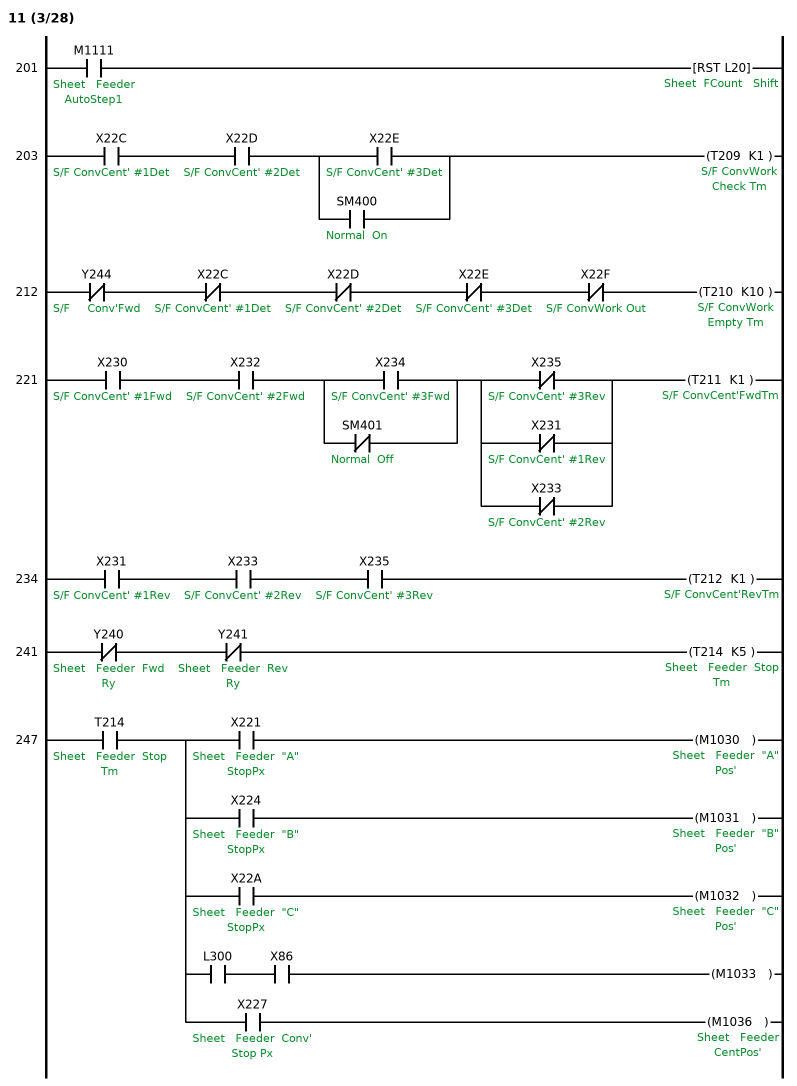
201   LD      M1111  ; Sheet   Feeder  AutoStep1
      RST     L20  ; Sheet  FCount   Shift
203   LD      X22C  ; S/F ConvCent' #1Det
      AND     X22D  ; S/F ConvCent' #2Det
      LD      X22E  ; S/F ConvCent' #3Det
      OR      SM400  ; Normal  On
      ANB
      OUT     T209 K1  ; S/F ConvWork    Check Tm
212   LDI     Y244  ; S/F     Conv'Fwd
      ANI     X22C  ; S/F ConvCent' #1Det
      ANI     X22D  ; S/F ConvCent' #2Det
      ANI     X22E  ; S/F ConvCent' #3Det
      ANI     X22F  ; S/F ConvWork Out
      OUT     T210 K10  ; S/F ConvWork    Empty Tm
221   LD      X230  ; S/F ConvCent' #1Fwd
      AND     X232  ; S/F ConvCent' #2Fwd
      LD      X234  ; S/F ConvCent' #3Fwd
      ORI     SM401  ; Normal  Off
      ANB
      LDI     X235  ; S/F ConvCent' #3Rev
      ORI     X231  ; S/F ConvCent' #1Rev
      ORI     X233  ; S/F ConvCent' #2Rev
      ANB
      OUT     T211 K1  ; S/F ConvCent'FwdTm
234   LD      X231  ; S/F ConvCent' #1Rev
      AND     X233  ; S/F ConvCent' #2Rev
      AND     X235  ; S/F ConvCent' #3Rev
      OUT     T212 K1  ; S/F ConvCent'RevTm
241   LDI     Y240  ; Sheet   Feeder  Fwd Ry
      ANI     Y241  ; Sheet   Feeder  Rev Ry
      OUT     T214 K5  ; Sheet   Feeder  Stop Tm
247   LD      T214  ; Sheet   Feeder  Stop Tm
      MPS
      AND     X221  ; Sheet   Feeder  "A" StopPx
      OUT     M1030  ; Sheet   Feeder  "A" Pos'
      MRD
      AND     X224  ; Sheet   Feeder  "B" StopPx
      OUT     M1031  ; Sheet   Feeder  "B" Pos'
      MRD
      AND     X22A  ; Sheet   Feeder  "C" StopPx
      OUT     M1032  ; Sheet   Feeder  "C" Pos'
      MRD
      AND     L300
      AND     X86
      OUT     M1033
      MPP
      AND     X227  ; Sheet   Feeder  Conv'   Stop Px
      OUT     M1036  ; Sheet   Feeder  CentPos'
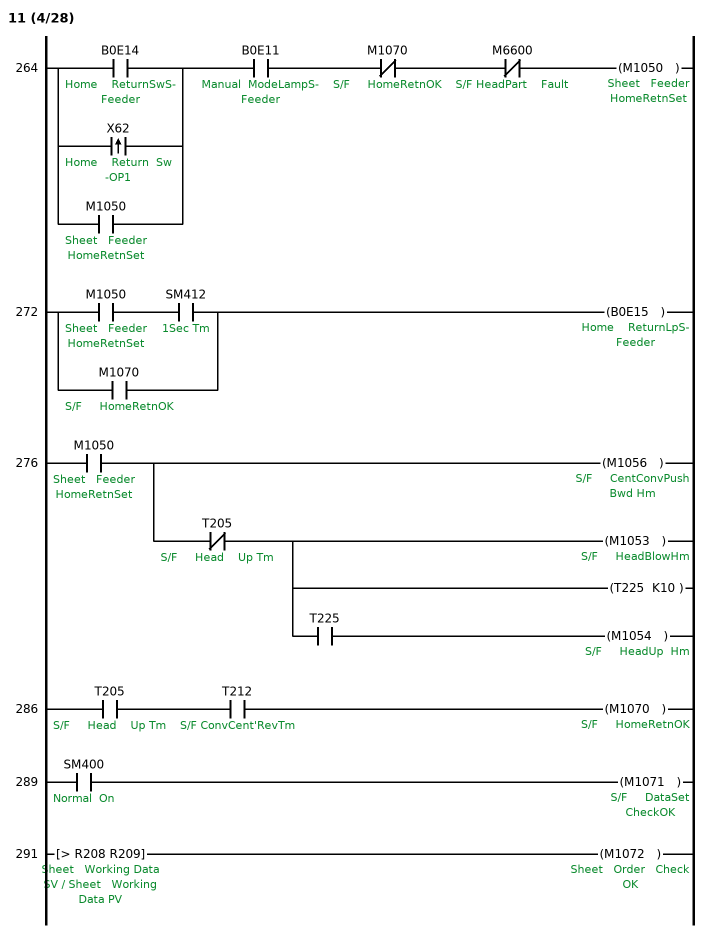
264   LD      B0E14  ; Home    ReturnSwS-Feeder
      ORP     X62  ; Home    Return  Sw -OP1
      OR      M1050  ; Sheet   Feeder  HomeRetnSet
      AND     B0E11  ; Manual  ModeLampS-Feeder
      ANI     M1070  ; S/F     HomeRetnOK
      ANI     M6600  ; S/F HeadPart    Fault
      OUT     M1050  ; Sheet   Feeder  HomeRetnSet
272   LD      M1050  ; Sheet   Feeder  HomeRetnSet
      AND     SM412  ; 1Sec Tm
      OR      M1070  ; S/F     HomeRetnOK
      OUT     B0E15  ; Home    ReturnLpS-Feeder
276   LD      M1050  ; Sheet   Feeder  HomeRetnSet
      OUT     M1056  ; S/F     CentConvPushBwd Hm
      ANI     T205  ; S/F     Head    Up Tm
      OUT     M1053  ; S/F     HeadBlowHm
      OUT     T225 K10
      AND     T225
      OUT     M1054  ; S/F     HeadUp  Hm
286   LD      T205  ; S/F     Head    Up Tm
      AND     T212  ; S/F ConvCent'RevTm
      OUT     M1070  ; S/F     HomeRetnOK
289   LD      SM400  ; Normal  On
      OUT     M1071  ; S/F     DataSet CheckOK
291   LD>     R208 R209  ; Sheet   Working Data SV / Sheet   Working Data PV
      OUT     M1072  ; Sheet   Order   Check OK
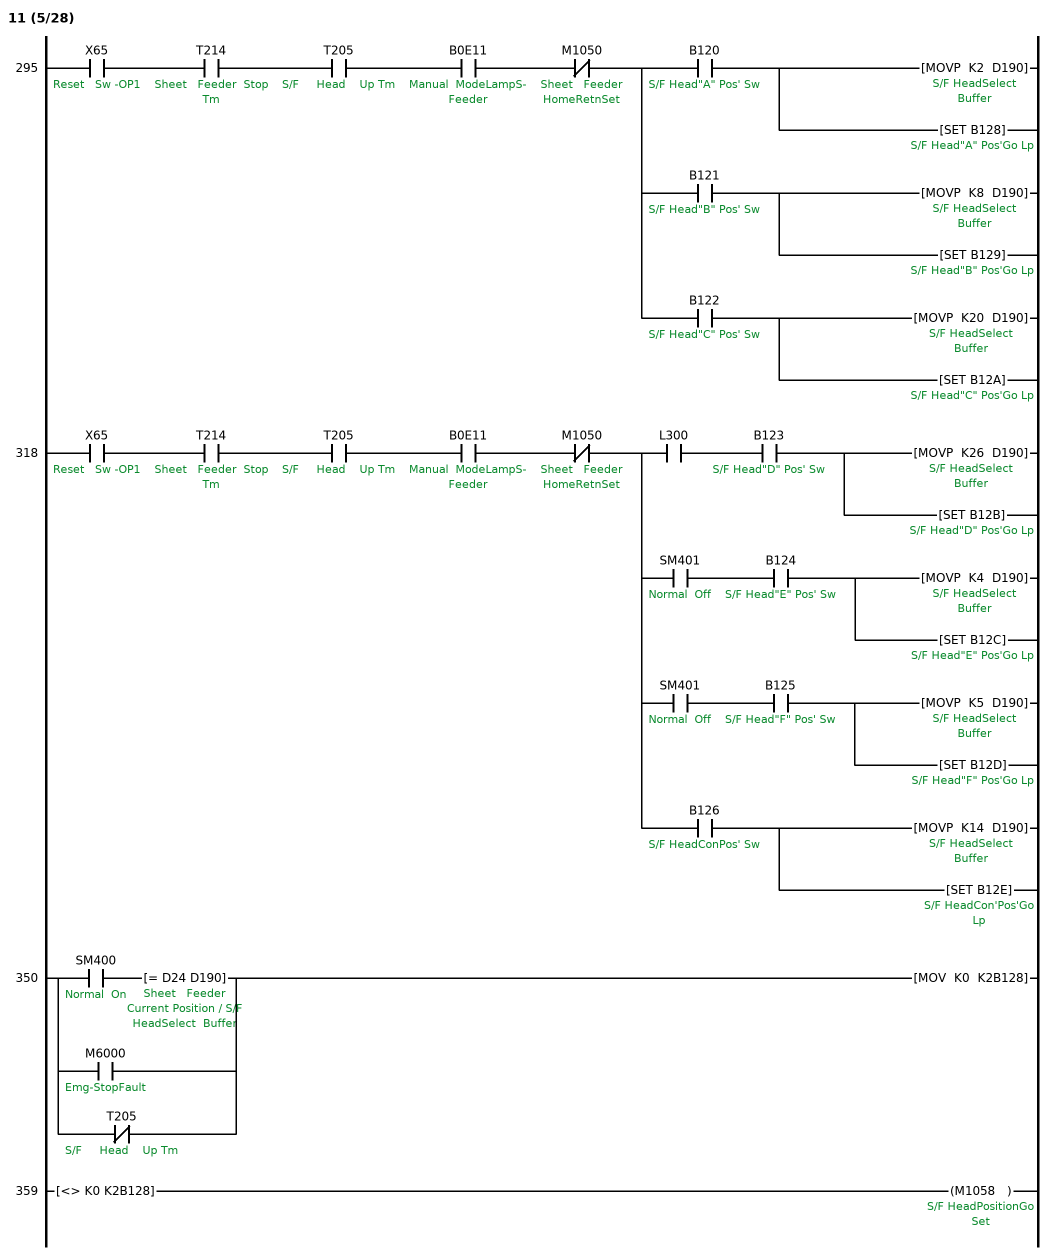
295   LD      X65  ; Reset   Sw -OP1
      AND     T214  ; Sheet   Feeder  Stop Tm
      AND     T205  ; S/F     Head    Up Tm
      AND     B0E11  ; Manual  ModeLampS-Feeder
      ANI     M1050  ; Sheet   Feeder  HomeRetnSet
      MPS
      AND     B120  ; S/F Head"A" Pos' Sw
      MOVP    K2 D190  ; S/F HeadSelect  Buffer
      SET     B128  ; S/F Head"A" Pos'Go Lp
      MRD
      AND     B121  ; S/F Head"B" Pos' Sw
      MOVP    K8 D190
      SET     B129  ; S/F Head"B" Pos'Go Lp
      MPP
      AND     B122  ; S/F Head"C" Pos' Sw
      MOVP    K20 D190
      SET     B12A  ; S/F Head"C" Pos'Go Lp
318   LD      X65  ; Reset   Sw -OP1
      AND     T214  ; Sheet   Feeder  Stop Tm
      AND     T205  ; S/F     Head    Up Tm
      AND     B0E11  ; Manual  ModeLampS-Feeder
      ANI     M1050  ; Sheet   Feeder  HomeRetnSet
      MPS
      AND     L300
      AND     B123  ; S/F Head"D" Pos' Sw
      MOVP    K26 D190
      SET     B12B  ; S/F Head"D" Pos'Go Lp
      MRD
      AND     SM401  ; Normal  Off
      AND     B124  ; S/F Head"E" Pos' Sw
      MOVP    K4 D190
      SET     B12C  ; S/F Head"E" Pos'Go Lp
      MRD
      AND     SM401  ; Normal  Off
      AND     B125  ; S/F Head"F" Pos' Sw
      MOVP    K5 D190
      SET     B12D  ; S/F Head"F" Pos'Go Lp
      MPP
      AND     B126  ; S/F HeadConPos' Sw
      MOVP    K14 D190
      SET     B12E  ; S/F HeadCon'Pos'Go Lp
350   LD      SM400  ; Normal  On
      AND=    D24 D190  ; Sheet   Feeder  Current Position / S/F HeadSelect  Buffer
      OR      M6000  ; Emg-StopFault
      ORI     T205  ; S/F     Head    Up Tm
      MOV     K0 K2B128
359   LD<>    K0 K2B128  ; S/F Head"A" Pos'Go Lp
      OUT     M1058  ; S/F HeadPositionGo Set
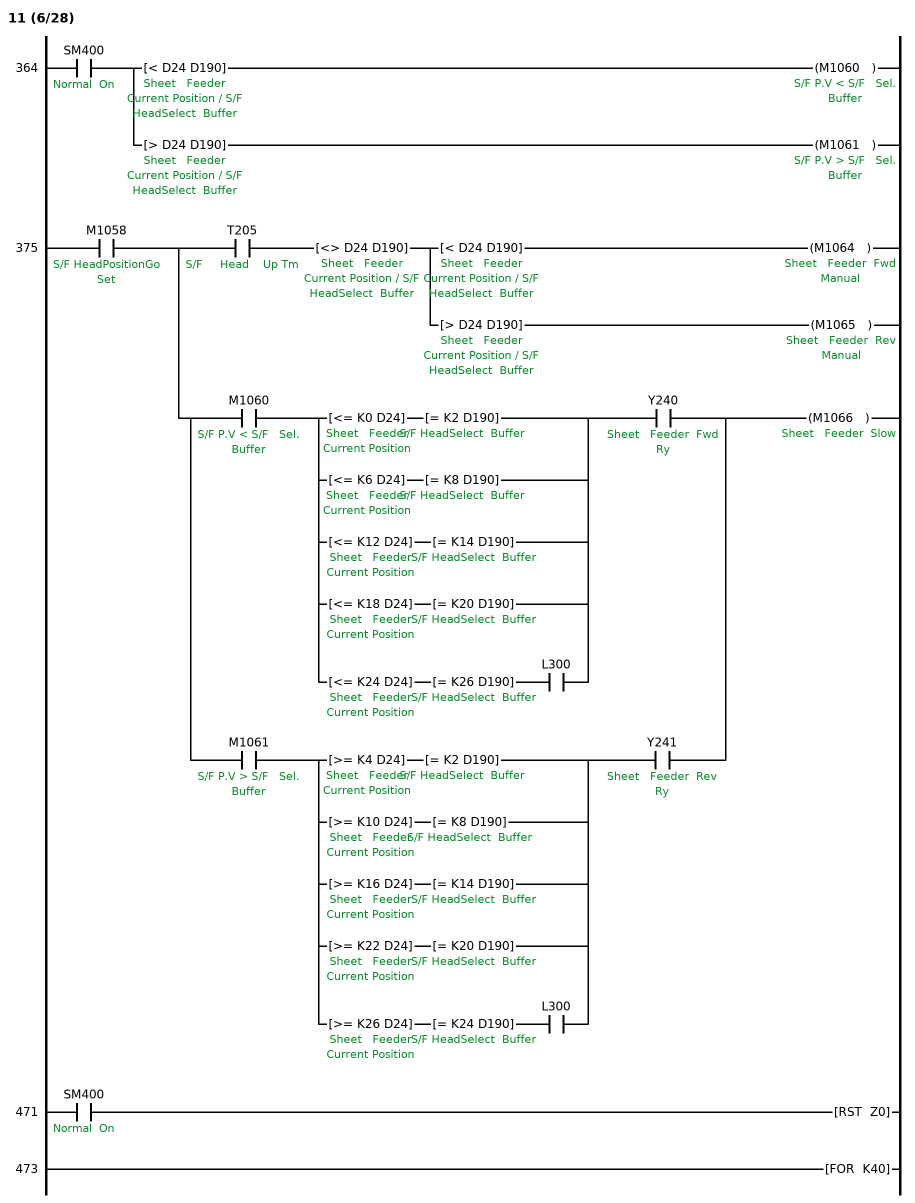
364   LD      SM400  ; Normal  On
      MPS
      AND<    D24 D190  ; Sheet   Feeder  Current Position / S/F HeadSelect  Buffer
      OUT     M1060  ; S/F P.V < S/F   Sel.    Buffer
      MPP
      AND>    D24 D190  ; Sheet   Feeder  Current Position / S/F HeadSelect  Buffer
      OUT     M1061  ; S/F P.V > S/F   Sel.    Buffer
375   LD      M1058  ; S/F HeadPositionGo Set
      MPS
      AND     T205  ; S/F     Head    Up Tm
      AND<>   D24 D190  ; Sheet   Feeder  Current Position / S/F HeadSelect  Buffer
      MPS
      AND<    D24 D190  ; Sheet   Feeder  Current Position / S/F HeadSelect  Buffer
      OUT     M1064  ; Sheet   Feeder  Fwd     Manual
      MPP
      AND>    D24 D190  ; Sheet   Feeder  Current Position / S/F HeadSelect  Buffer
      OUT     M1065  ; Sheet   Feeder  Rev     Manual
      MPP
      LD      M1060  ; S/F P.V < S/F   Sel.    Buffer
      LD<=    K0 D24  ; Sheet   Feeder  Current Position
      AND=    K2 D190  ; S/F HeadSelect  Buffer
      LD<=    K6 D24  ; Sheet   Feeder  Current Position
      AND=    K8 D190  ; S/F HeadSelect  Buffer
      ORB
      LD<=    K12 D24  ; Sheet   Feeder  Current Position
      AND=    K14 D190  ; S/F HeadSelect  Buffer
      ORB
      LD<=    K18 D24  ; Sheet   Feeder  Current Position
      AND=    K20 D190  ; S/F HeadSelect  Buffer
      ORB
      LD<=    K24 D24  ; Sheet   Feeder  Current Position
      AND=    K26 D190  ; S/F HeadSelect  Buffer
      AND     L300
      ORB
      ANB
      AND     Y240  ; Sheet   Feeder  Fwd Ry
      LD      M1061  ; S/F P.V > S/F   Sel.    Buffer
      LD>=    K4 D24  ; Sheet   Feeder  Current Position
      AND=    K2 D190  ; S/F HeadSelect  Buffer
      LD>=    K10 D24  ; Sheet   Feeder  Current Position
      AND=    K8 D190  ; S/F HeadSelect  Buffer
      ORB
      LD>=    K16 D24  ; Sheet   Feeder  Current Position
      AND=    K14 D190  ; S/F HeadSelect  Buffer
      ORB
      LD>=    K22 D24  ; Sheet   Feeder  Current Position
      AND=    K20 D190  ; S/F HeadSelect  Buffer
      ORB
      LD>=    K26 D24  ; Sheet   Feeder  Current Position
      AND=    K24 D190  ; S/F HeadSelect  Buffer
      AND     L300
      ORB
      ANB
      AND     Y241  ; Sheet   Feeder  Rev Ry
      ORB
      ANB
      OUT     M1066  ; Sheet   Feeder  Slow
471   LD      SM400  ; Normal  On
      RST     Z0
473   FOR     K40
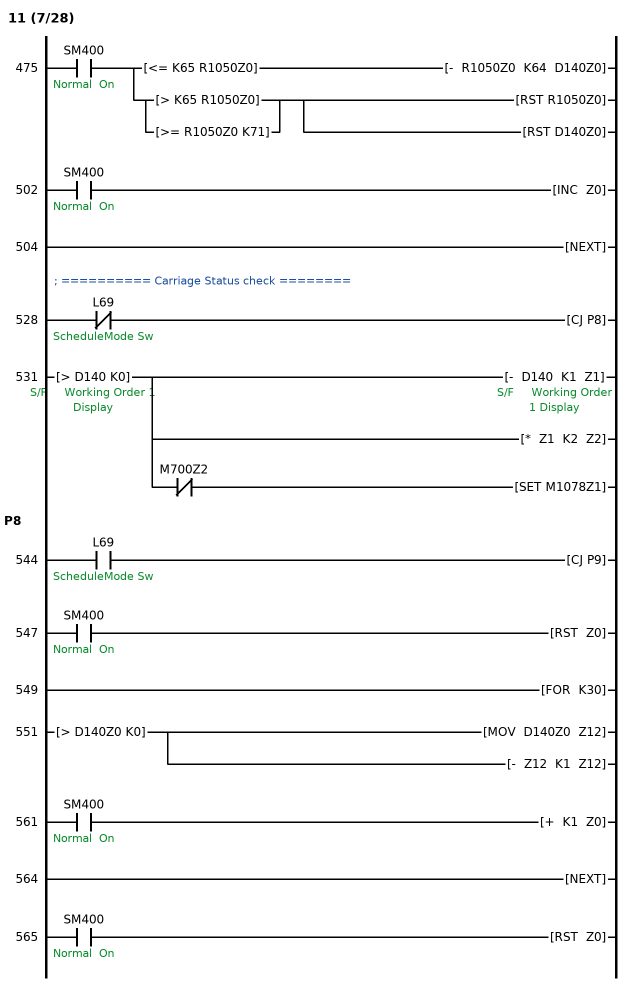
475   LD      SM400  ; Normal  On
      MPS
      AND<=   K65 R1050Z0
      -       R1050Z0 K64 D140Z0
      MPP
      LD>     K65 R1050Z0
      OR>=    R1050Z0 K71
      ANB
      RST     R1050Z0
      RST     D140Z0
502   LD      SM400  ; Normal  On
      INC     Z0
504   NEXT
; ========== Carriage Status check ========
528   LDI     L69  ; ScheduleMode Sw
      CJ      P8
531   LD>     D140 K0  ; S/F     Working Order 1 Display
      -       D140 K1 Z1
      *       Z1 K2 Z2
      ANI     M700Z2
      SET     M1078Z1
      P8
544   LD      L69  ; ScheduleMode Sw
      CJ      P9
547   LD      SM400  ; Normal  On
      RST     Z0
549   FOR     K30
551   LD>     D140Z0 K0
      MOV     D140Z0 Z12
      -       Z12 K1 Z12
561   LD      SM400  ; Normal  On
      +       K1 Z0
564   NEXT
565   LD      SM400  ; Normal  On
      RST     Z0
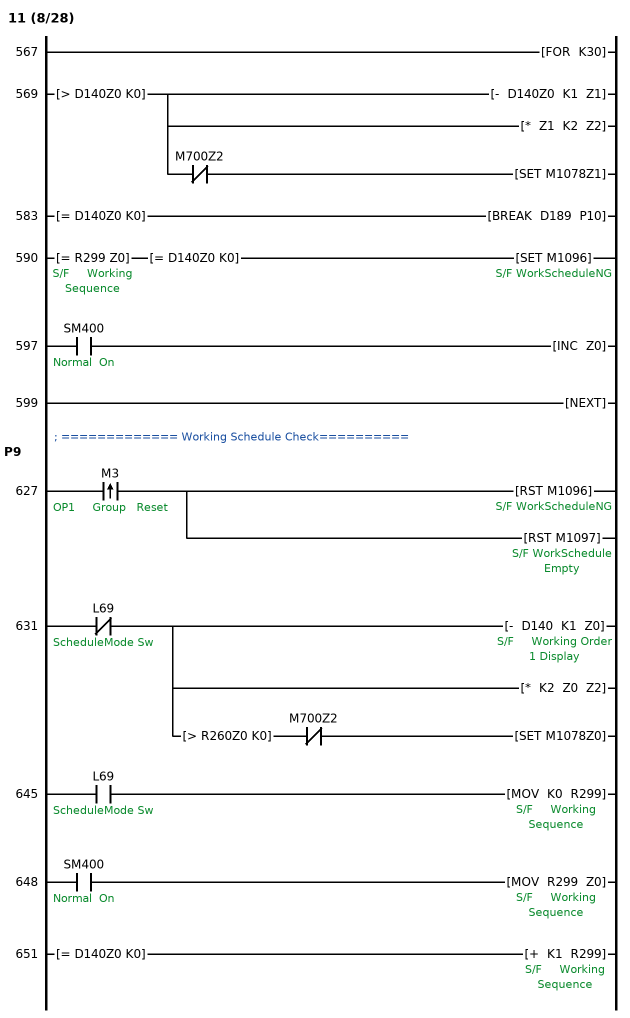
567   FOR     K30
569   LD>     D140Z0 K0
      -       D140Z0 K1 Z1
      *       Z1 K2 Z2
      ANI     M700Z2
      SET     M1078Z1
583   LD=     D140Z0 K0
      BREAK   D189 P10
590   LD=     R299 Z0  ; S/F     Working Sequence
      AND=    D140Z0 K0
      SET     M1096  ; S/F WorkScheduleNG
597   LD      SM400  ; Normal  On
      INC     Z0
599   NEXT
      P10
; ============= Working Schedule Check==========
      P9
627   LDP     M3  ; OP1     Group   Reset
      RST     M1096  ; S/F WorkScheduleNG
      RST     M1097  ; S/F WorkScheduleEmpty
631   LDI     L69  ; ScheduleMode Sw
      -       D140 K1 Z0
      *       K2 Z0 Z2
      AND>    R260Z0 K0
      ANI     M700Z2
      SET     M1078Z0
645   LD      L69  ; ScheduleMode Sw
      MOV     K0 R299
648   LD      SM400  ; Normal  On
      MOV     R299 Z0
651   LD=     D140Z0 K0
      +       K1 R299
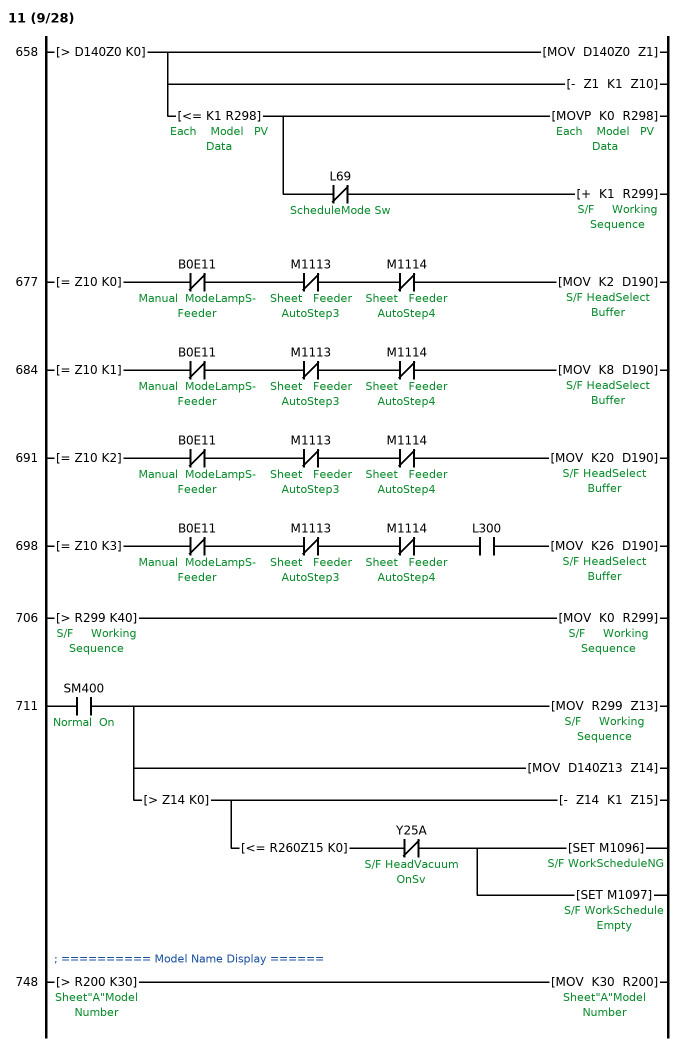
658   LD>     D140Z0 K0
      MOV     D140Z0 Z1
      -       Z1 K1 Z10
      AND<=   K1 R298  ; Each    Model   PV Data
      MOVP    K0 R298
      ANI     L69  ; ScheduleMode Sw
      +       K1 R299
677   LD=     Z10 K0
      ANI     B0E11  ; Manual  ModeLampS-Feeder
      ANI     M1113  ; Sheet   Feeder  AutoStep3
      ANI     M1114  ; Sheet   Feeder  AutoStep4
      MOV     K2 D190
684   LD=     Z10 K1
      ANI     B0E11  ; Manual  ModeLampS-Feeder
      ANI     M1113  ; Sheet   Feeder  AutoStep3
      ANI     M1114  ; Sheet   Feeder  AutoStep4
      MOV     K8 D190
691   LD=     Z10 K2
      ANI     B0E11  ; Manual  ModeLampS-Feeder
      ANI     M1113  ; Sheet   Feeder  AutoStep3
      ANI     M1114  ; Sheet   Feeder  AutoStep4
      MOV     K20 D190
698   LD=     Z10 K3
      ANI     B0E11  ; Manual  ModeLampS-Feeder
      ANI     M1113  ; Sheet   Feeder  AutoStep3
      ANI     M1114  ; Sheet   Feeder  AutoStep4
      AND     L300
      MOV     K26 D190
706   LD>     R299 K40  ; S/F     Working Sequence
      MOV     K0 R299
711   LD      SM400  ; Normal  On
      MOV     R299 Z13
      MOV     D140Z13 Z14
      AND>    Z14 K0
      -       Z14 K1 Z15
      AND<=   R260Z15 K0
      ANI     Y25A  ; S/F HeadVacuum  OnSv
      SET     M1096  ; S/F WorkScheduleNG
      SET     M1097  ; S/F WorkScheduleEmpty
; ========== Model Name Display ======
748   LD>     R200 K30  ; Sheet"A"Model   Number
      MOV     K30 R200
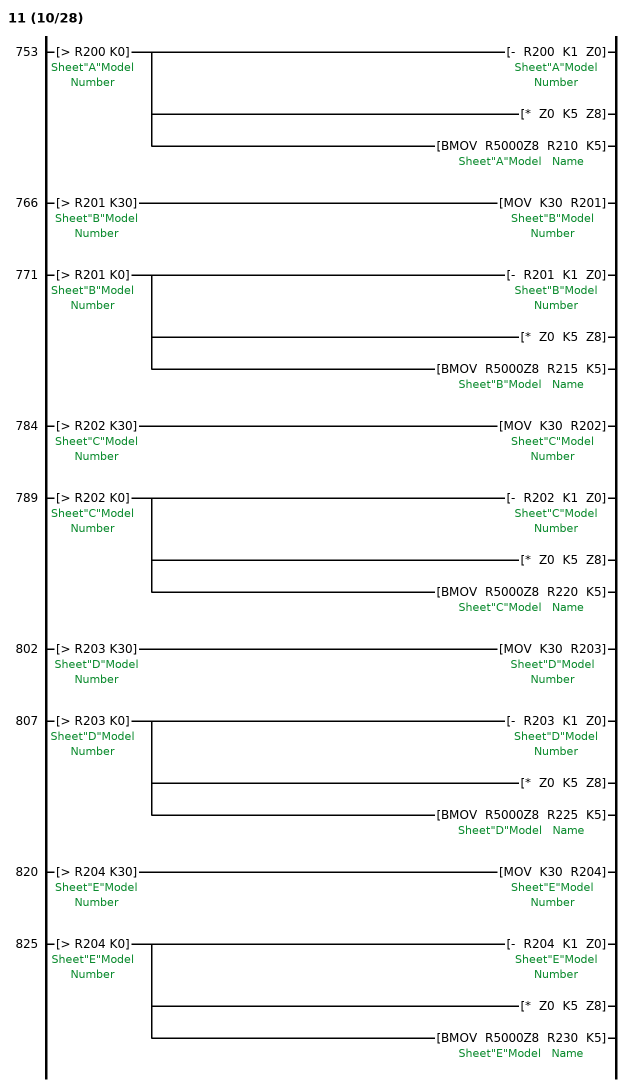
753   LD>     R200 K0  ; Sheet"A"Model   Number
      -       R200 K1 Z0
      *       Z0 K5 Z8
      BMOV    R5000Z8 R210 K5  ; Sheet"A"Model   Name
766   LD>     R201 K30  ; Sheet"B"Model   Number
      MOV     K30 R201
771   LD>     R201 K0  ; Sheet"B"Model   Number
      -       R201 K1 Z0
      *       Z0 K5 Z8
      BMOV    R5000Z8 R215 K5  ; Sheet"B"Model   Name
784   LD>     R202 K30  ; Sheet"C"Model   Number
      MOV     K30 R202
789   LD>     R202 K0  ; Sheet"C"Model   Number
      -       R202 K1 Z0
      *       Z0 K5 Z8
      BMOV    R5000Z8 R220 K5  ; Sheet"C"Model   Name
802   LD>     R203 K30  ; Sheet"D"Model   Number
      MOV     K30 R203
807   LD>     R203 K0  ; Sheet"D"Model   Number
      -       R203 K1 Z0
      *       Z0 K5 Z8
      BMOV    R5000Z8 R225 K5  ; Sheet"D"Model   Name
820   LD>     R204 K30  ; Sheet"E"Model   Number
      MOV     K30 R204
825   LD>     R204 K0  ; Sheet"E"Model   Number
      -       R204 K1 Z0
      *       Z0 K5 Z8
      BMOV    R5000Z8 R230 K5  ; Sheet"E"Model   Name
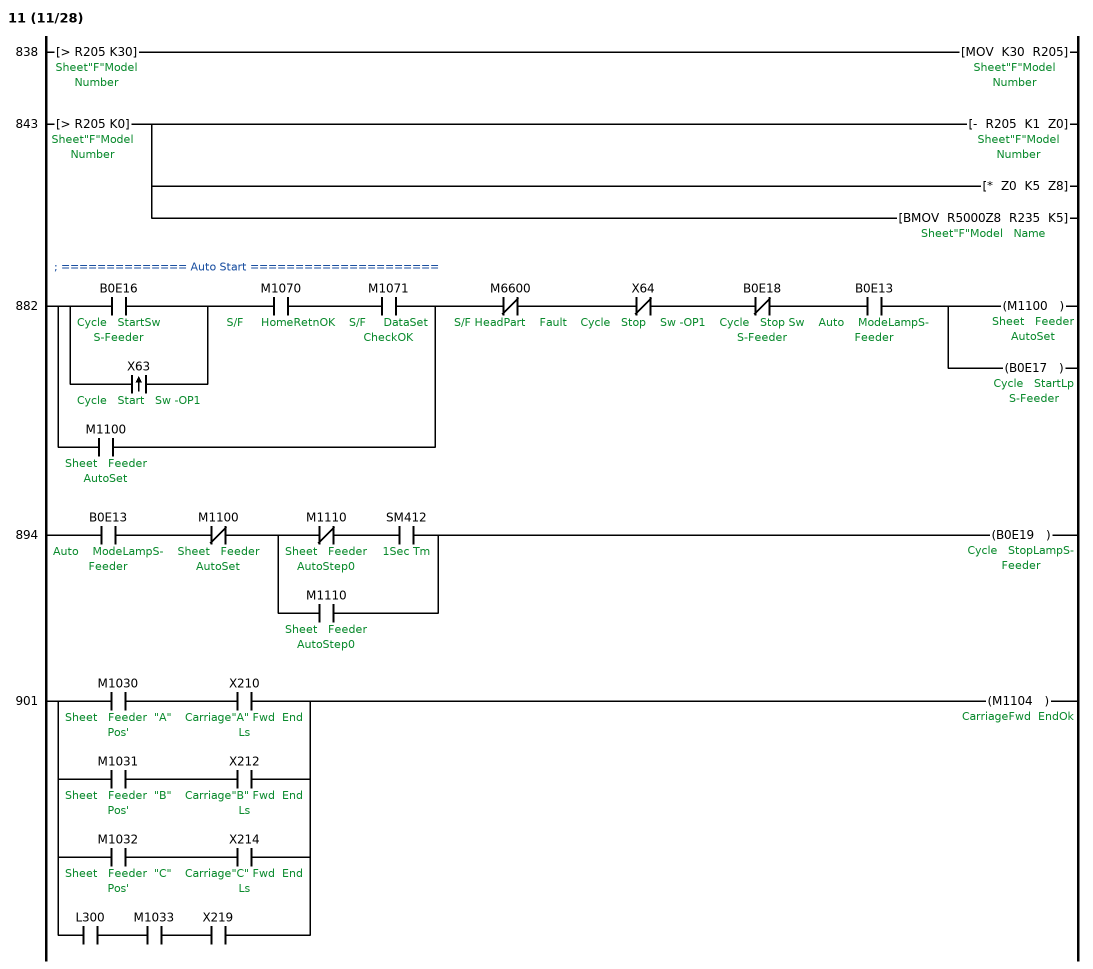
838   LD>     R205 K30  ; Sheet"F"Model   Number
      MOV     K30 R205
843   LD>     R205 K0  ; Sheet"F"Model   Number
      -       R205 K1 Z0
      *       Z0 K5 Z8
      BMOV    R5000Z8 R235 K5  ; Sheet"F"Model   Name
; ============== Auto Start =====================
882   LD      B0E16  ; Cycle   StartSw S-Feeder
      ORP     X63  ; Cycle   Start   Sw -OP1
      AND     M1070  ; S/F     HomeRetnOK
      AND     M1071  ; S/F     DataSet CheckOK
      OR      M1100  ; Sheet   Feeder  AutoSet
      ANI     M6600  ; S/F HeadPart    Fault
      ANI     X64  ; Cycle   Stop    Sw -OP1
      ANI     B0E18  ; Cycle   Stop Sw S-Feeder
      AND     B0E13  ; Auto    ModeLampS-Feeder
      OUT     M1100  ; Sheet   Feeder  AutoSet
      OUT     B0E17  ; Cycle   StartLp S-Feeder
894   LD      B0E13  ; Auto    ModeLampS-Feeder
      ANI     M1100  ; Sheet   Feeder  AutoSet
      LDI     M1110  ; Sheet   Feeder  AutoStep0
      AND     SM412  ; 1Sec Tm
      OR      M1110  ; Sheet   Feeder  AutoStep0
      ANB
      OUT     B0E19  ; Cycle   StopLampS-Feeder
901   LD      M1030  ; Sheet   Feeder  "A" Pos'
      AND     X210  ; Carriage"A" Fwd  End Ls
      LD      M1031  ; Sheet   Feeder  "B" Pos'
      AND     X212  ; Carriage"B" Fwd  End Ls
      ORB
      LD      M1032  ; Sheet   Feeder  "C" Pos'
      AND     X214  ; Carriage"C" Fwd  End Ls
      ORB
      LD      L300
      AND     M1033
      AND     X219
      ORB
      OUT     M1104  ; CarriageFwd  EndOk
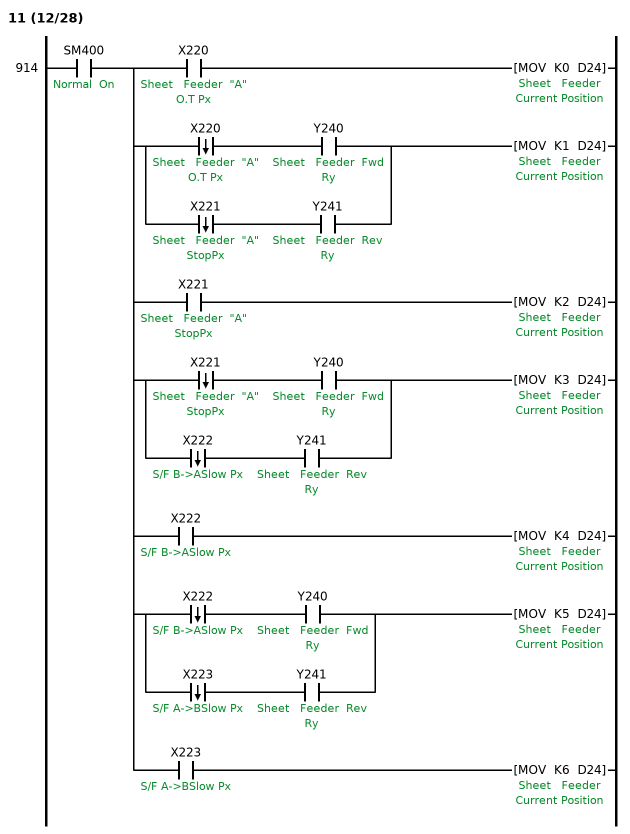
914   LD      SM400  ; Normal  On
      MPS
      AND     X220  ; Sheet   Feeder  "A" O.T Px
      MOV     K0 D24
      MRD
      LDF     X220  ; Sheet   Feeder  "A" O.T Px
      AND     Y240  ; Sheet   Feeder  Fwd Ry
      LDF     X221  ; Sheet   Feeder  "A" StopPx
      AND     Y241  ; Sheet   Feeder  Rev Ry
      ORB
      ANB
      MOV     K1 D24
      MRD
      AND     X221  ; Sheet   Feeder  "A" StopPx
      MOV     K2 D24
      MRD
      LDF     X221  ; Sheet   Feeder  "A" StopPx
      AND     Y240  ; Sheet   Feeder  Fwd Ry
      LDF     X222  ; S/F B->ASlow Px
      AND     Y241  ; Sheet   Feeder  Rev Ry
      ORB
      ANB
      MOV     K3 D24
      MRD
      AND     X222  ; S/F B->ASlow Px
      MOV     K4 D24
      MRD
      LDF     X222  ; S/F B->ASlow Px
      AND     Y240  ; Sheet   Feeder  Fwd Ry
      LDF     X223  ; S/F A->BSlow Px
      AND     Y241  ; Sheet   Feeder  Rev Ry
      ORB
      ANB
      MOV     K5 D24
      MPP
      AND     X223  ; S/F A->BSlow Px
      MOV     K6 D24
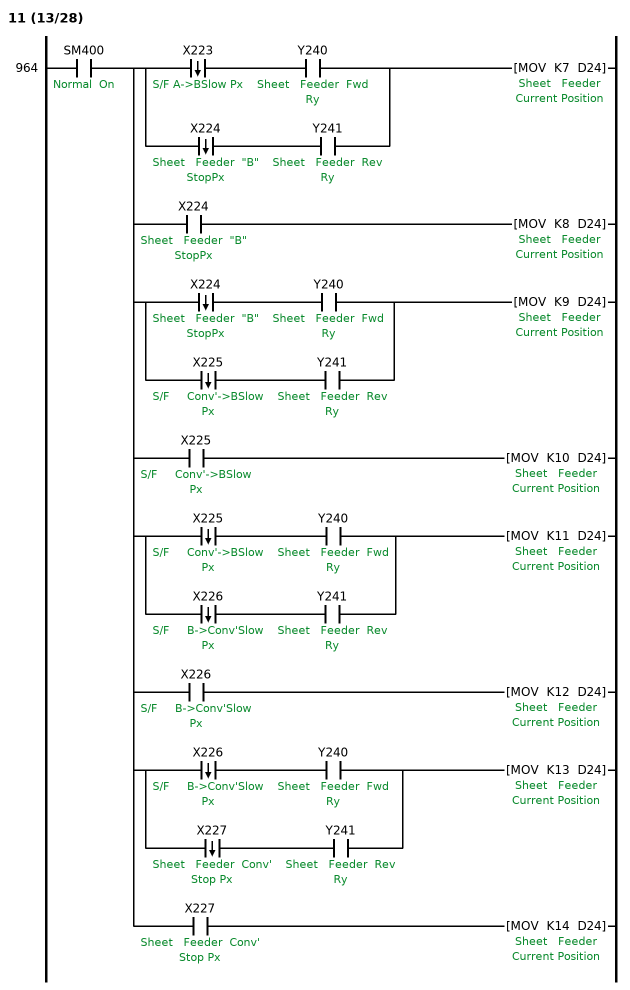
964   LD      SM400  ; Normal  On
      MPS
      LDF     X223  ; S/F A->BSlow Px
      AND     Y240  ; Sheet   Feeder  Fwd Ry
      LDF     X224  ; Sheet   Feeder  "B" StopPx
      AND     Y241  ; Sheet   Feeder  Rev Ry
      ORB
      ANB
      MOV     K7 D24
      MRD
      AND     X224  ; Sheet   Feeder  "B" StopPx
      MOV     K8 D24
      MRD
      LDF     X224  ; Sheet   Feeder  "B" StopPx
      AND     Y240  ; Sheet   Feeder  Fwd Ry
      LDF     X225  ; S/F     Conv'->BSlow Px
      AND     Y241  ; Sheet   Feeder  Rev Ry
      ORB
      ANB
      MOV     K9 D24
      MRD
      AND     X225  ; S/F     Conv'->BSlow Px
      MOV     K10 D24
      MRD
      LDF     X225  ; S/F     Conv'->BSlow Px
      AND     Y240  ; Sheet   Feeder  Fwd Ry
      LDF     X226  ; S/F     B->Conv'Slow Px
      AND     Y241  ; Sheet   Feeder  Rev Ry
      ORB
      ANB
      MOV     K11 D24
      MRD
      AND     X226  ; S/F     B->Conv'Slow Px
      MOV     K12 D24
      MRD
      LDF     X226  ; S/F     B->Conv'Slow Px
      AND     Y240  ; Sheet   Feeder  Fwd Ry
      LDF     X227  ; Sheet   Feeder  Conv'   Stop Px
      AND     Y241  ; Sheet   Feeder  Rev Ry
      ORB
      ANB
      MOV     K13 D24
      MPP
      AND     X227  ; Sheet   Feeder  Conv'   Stop Px
      MOV     K14 D24
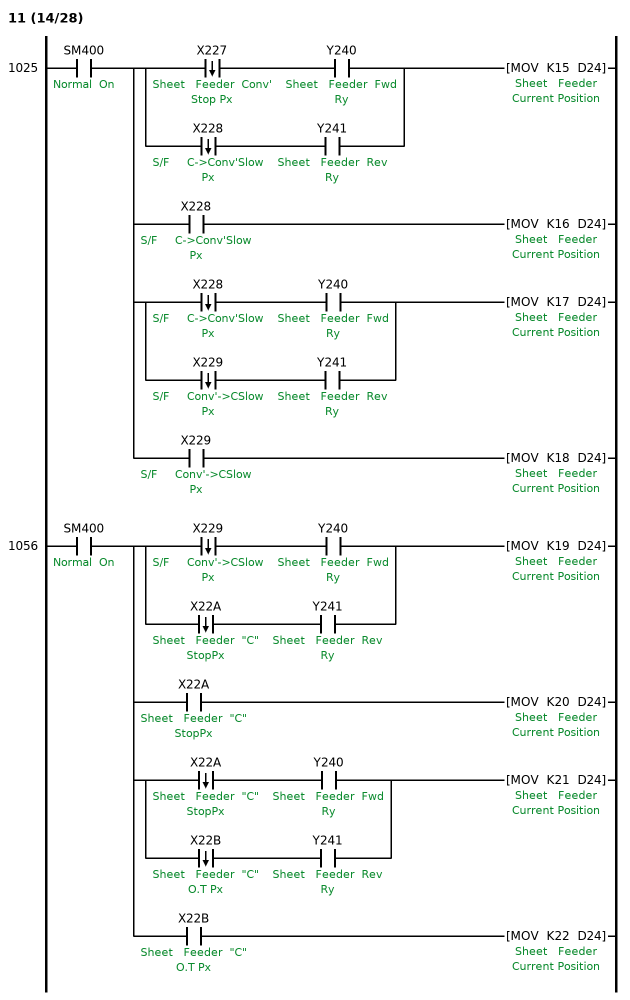
1025  LD      SM400  ; Normal  On
      MPS
      LDF     X227  ; Sheet   Feeder  Conv'   Stop Px
      AND     Y240  ; Sheet   Feeder  Fwd Ry
      LDF     X228  ; S/F     C->Conv'Slow Px
      AND     Y241  ; Sheet   Feeder  Rev Ry
      ORB
      ANB
      MOV     K15 D24
      MRD
      AND     X228  ; S/F     C->Conv'Slow Px
      MOV     K16 D24
      MRD
      LDF     X228  ; S/F     C->Conv'Slow Px
      AND     Y240  ; Sheet   Feeder  Fwd Ry
      LDF     X229  ; S/F     Conv'->CSlow Px
      AND     Y241  ; Sheet   Feeder  Rev Ry
      ORB
      ANB
      MOV     K17 D24
      MPP
      AND     X229  ; S/F     Conv'->CSlow Px
      MOV     K18 D24
1056  LD      SM400  ; Normal  On
      MPS
      LDF     X229  ; S/F     Conv'->CSlow Px
      AND     Y240  ; Sheet   Feeder  Fwd Ry
      LDF     X22A  ; Sheet   Feeder  "C" StopPx
      AND     Y241  ; Sheet   Feeder  Rev Ry
      ORB
      ANB
      MOV     K19 D24
      MRD
      AND     X22A  ; Sheet   Feeder  "C" StopPx
      MOV     K20 D24
      MRD
      LDF     X22A  ; Sheet   Feeder  "C" StopPx
      AND     Y240  ; Sheet   Feeder  Fwd Ry
      LDF     X22B  ; Sheet   Feeder  "C" O.T Px
      AND     Y241  ; Sheet   Feeder  Rev Ry
      ORB
      ANB
      MOV     K21 D24
      MPP
      AND     X22B  ; Sheet   Feeder  "C" O.T Px
      MOV     K22 D24
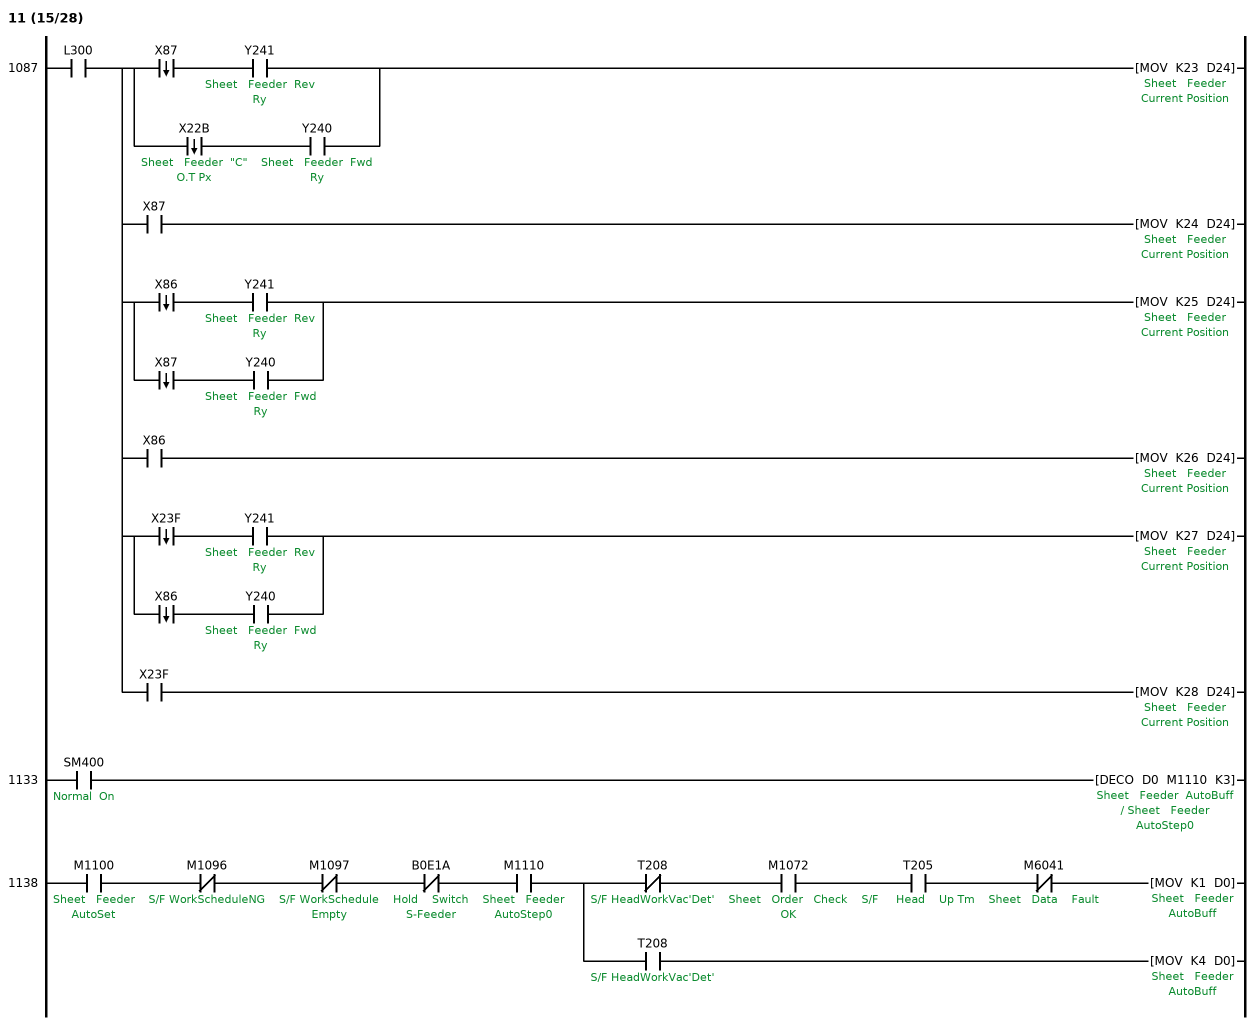
1087  LD      L300
      MPS
      LDF     X87
      AND     Y241  ; Sheet   Feeder  Rev Ry
      LDF     X22B  ; Sheet   Feeder  "C" O.T Px
      AND     Y240  ; Sheet   Feeder  Fwd Ry
      ORB
      ANB
      MOV     K23 D24
      MRD
      AND     X87
      MOV     K24 D24
      MRD
      LDF     X86
      AND     Y241  ; Sheet   Feeder  Rev Ry
      LDF     X87
      AND     Y240  ; Sheet   Feeder  Fwd Ry
      ORB
      ANB
      MOV     K25 D24
      MRD
      AND     X86
      MOV     K26 D24
      MRD
      LDF     X23F
      AND     Y241  ; Sheet   Feeder  Rev Ry
      LDF     X86
      AND     Y240  ; Sheet   Feeder  Fwd Ry
      ORB
      ANB
      MOV     K27 D24
      MPP
      AND     X23F
      MOV     K28 D24
1133  LD      SM400  ; Normal  On
      DECO    D0 M1110 K3  ; Sheet   Feeder  AutoBuff
1138  LD      M1100  ; Sheet   Feeder  AutoSet
      ANI     M1096  ; S/F WorkScheduleNG
      ANI     M1097  ; S/F WorkScheduleEmpty
      ANI     B0E1A  ; Hold    Switch  S-Feeder
      AND     M1110  ; Sheet   Feeder  AutoStep0
      MPS
      ANI     T208  ; S/F HeadWorkVac'Det'
      AND     M1072  ; Sheet   Order   Check OK
      AND     T205  ; S/F     Head    Up Tm
      ANI     M6041  ; Sheet   Data    Fault
      MOV     K1 D0
      MPP
      AND     T208  ; S/F HeadWorkVac'Det'
      MOV     K4 D0
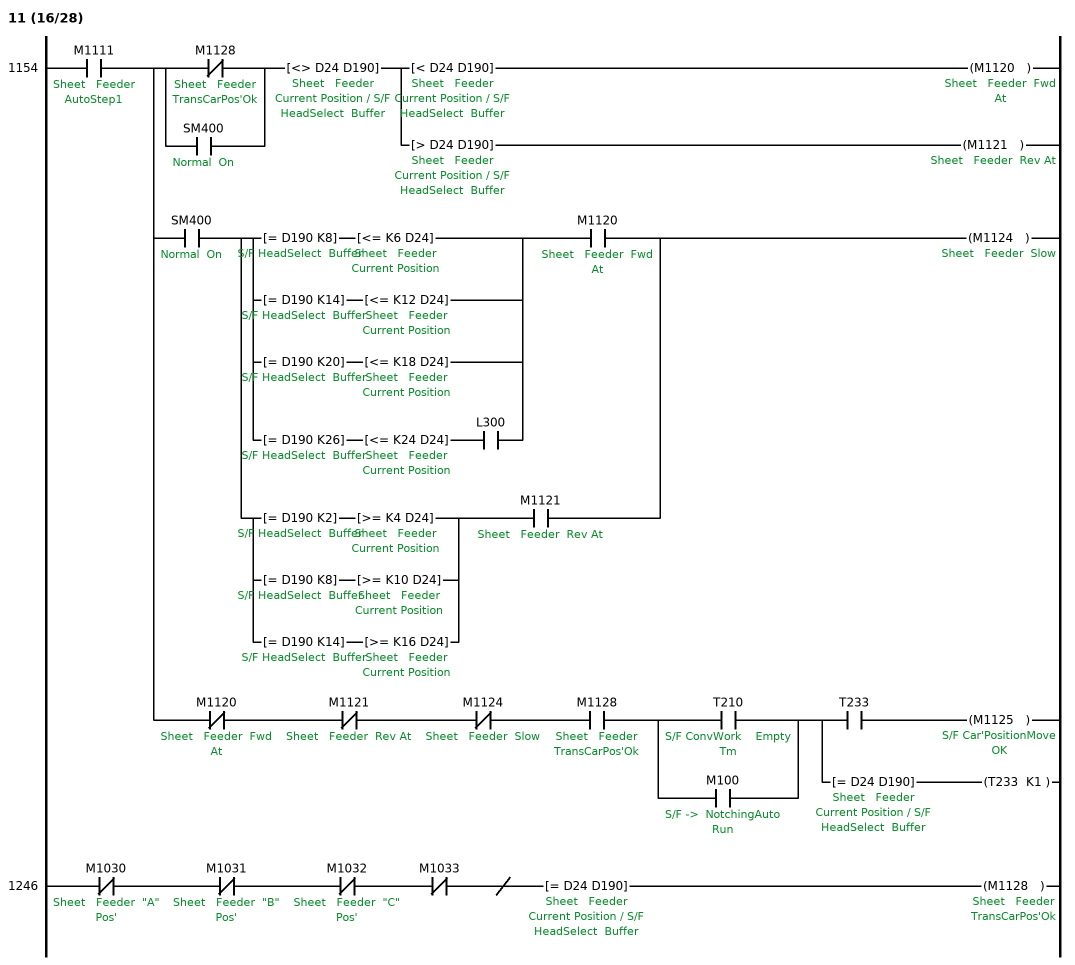
1154  LD      M1111  ; Sheet   Feeder  AutoStep1
      MPS
      LDI     M1128  ; Sheet   Feeder  TransCarPos'Ok
      OR      SM400  ; Normal  On
      ANB
      AND<>   D24 D190  ; Sheet   Feeder  Current Position / S/F HeadSelect  Buffer
      MPS
      AND<    D24 D190  ; Sheet   Feeder  Current Position / S/F HeadSelect  Buffer
      OUT     M1120  ; Sheet   Feeder  Fwd At
      MPP
      AND>    D24 D190  ; Sheet   Feeder  Current Position / S/F HeadSelect  Buffer
      OUT     M1121  ; Sheet   Feeder  Rev At
      MRD
      AND     SM400  ; Normal  On
      LD=     D190 K8  ; S/F HeadSelect  Buffer
      AND<=   K6 D24  ; Sheet   Feeder  Current Position
      LD=     D190 K14  ; S/F HeadSelect  Buffer
      AND<=   K12 D24  ; Sheet   Feeder  Current Position
      ORB
      LD=     D190 K20  ; S/F HeadSelect  Buffer
      AND<=   K18 D24  ; Sheet   Feeder  Current Position
      ORB
      LD=     D190 K26  ; S/F HeadSelect  Buffer
      AND<=   K24 D24  ; Sheet   Feeder  Current Position
      AND     L300
      ORB
      AND     M1120  ; Sheet   Feeder  Fwd At
      LD=     D190 K2  ; S/F HeadSelect  Buffer
      AND>=   K4 D24  ; Sheet   Feeder  Current Position
      LD=     D190 K8  ; S/F HeadSelect  Buffer
      AND>=   K10 D24  ; Sheet   Feeder  Current Position
      ORB
      LD=     D190 K14  ; S/F HeadSelect  Buffer
      AND>=   K16 D24  ; Sheet   Feeder  Current Position
      ORB
      AND     M1121  ; Sheet   Feeder  Rev At
      ORB
      ANB
      OUT     M1124  ; Sheet   Feeder  Slow
      MPP
      ANI     M1120  ; Sheet   Feeder  Fwd At
      ANI     M1121  ; Sheet   Feeder  Rev At
      ANI     M1124  ; Sheet   Feeder  Slow
      AND     M1128  ; Sheet   Feeder  TransCarPos'Ok
      LD      T210  ; S/F ConvWork    Empty Tm
      OR      M100  ; S/F ->  NotchingAuto Run
      ANB
      MPS
      AND     T233
      OUT     M1125  ; S/F Car'PositionMoveOK
      MPP
      AND=    D24 D190  ; Sheet   Feeder  Current Position / S/F HeadSelect  Buffer
      OUT     T233 K1
1246  LDI     M1030  ; Sheet   Feeder  "A" Pos'
      ANI     M1031  ; Sheet   Feeder  "B" Pos'
      ANI     M1032  ; Sheet   Feeder  "C" Pos'
      ANI     M1033
      INV
      AND=    D24 D190  ; Sheet   Feeder  Current Position / S/F HeadSelect  Buffer
      OUT     M1128  ; Sheet   Feeder  TransCarPos'Ok
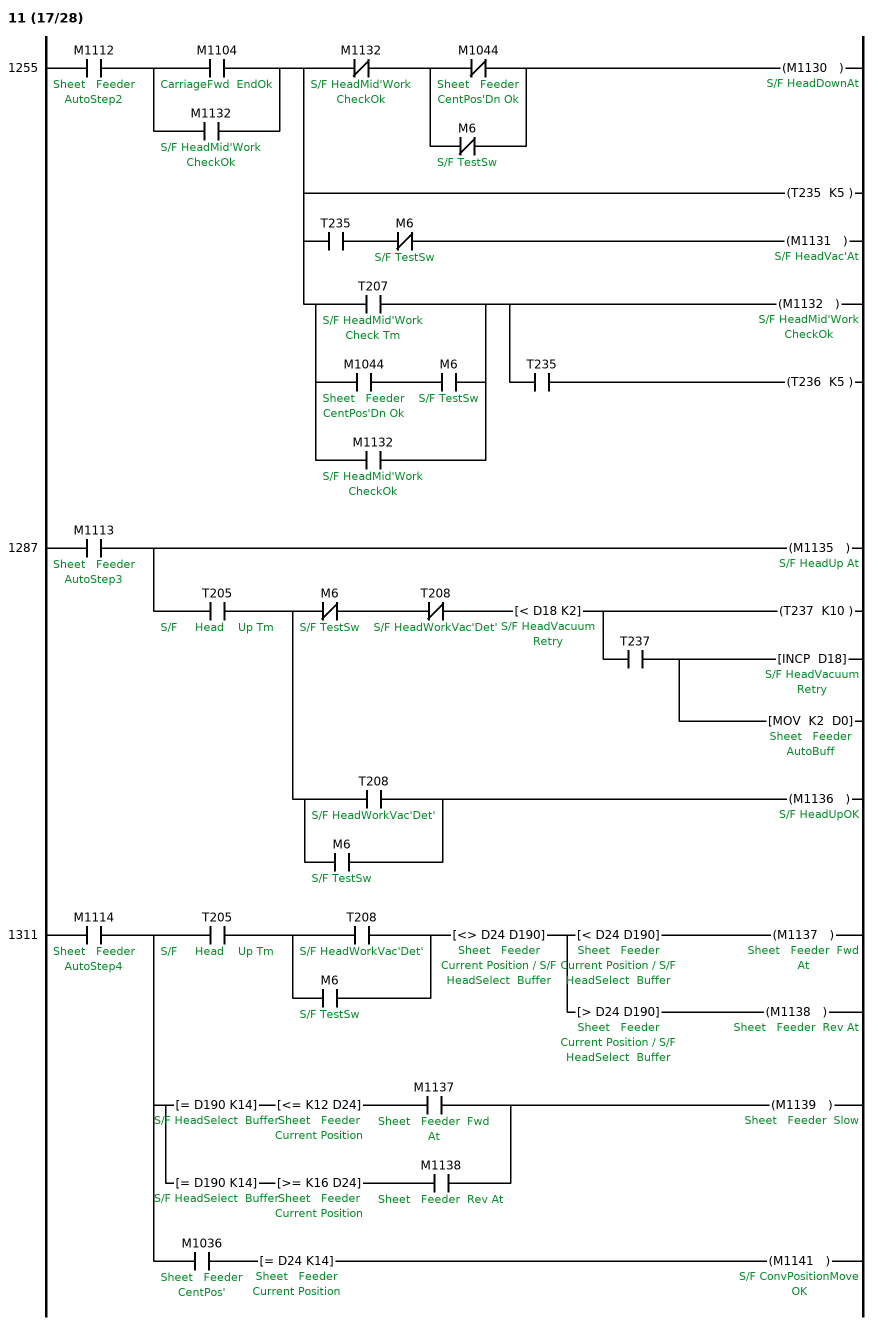
1255  LD      M1112  ; Sheet   Feeder  AutoStep2
      LD      M1104  ; CarriageFwd  EndOk
      OR      M1132  ; S/F HeadMid'WorkCheckOk
      ANB
      MPS
      ANI     M1132  ; S/F HeadMid'WorkCheckOk
      LDI     M1044  ; Sheet   Feeder  CentPos'Dn Ok
      ORI     M6  ; S/F TestSw
      ANB
      OUT     M1130  ; S/F HeadDownAt
      MPP
      OUT     T235 K5
      MPS
      AND     T235
      ANI     M6  ; S/F TestSw
      OUT     M1131  ; S/F HeadVac'At
      MPP
      LD      T207  ; S/F HeadMid'WorkCheck Tm
      LD      M1044  ; Sheet   Feeder  CentPos'Dn Ok
      AND     M6  ; S/F TestSw
      ORB
      OR      M1132  ; S/F HeadMid'WorkCheckOk
      ANB
      OUT     M1132  ; S/F HeadMid'WorkCheckOk
      AND     T235
      OUT     T236 K5
1287  LD      M1113  ; Sheet   Feeder  AutoStep3
      OUT     M1135  ; S/F HeadUp At
      AND     T205  ; S/F     Head    Up Tm
      MPS
      ANI     M6  ; S/F TestSw
      ANI     T208  ; S/F HeadWorkVac'Det'
      AND<    D18 K2  ; S/F HeadVacuum  Retry
      OUT     T237 K10
      AND     T237
      INCP    D18
      MOV     K2 D0
      MPP
      LD      T208  ; S/F HeadWorkVac'Det'
      OR      M6  ; S/F TestSw
      ANB
      OUT     M1136  ; S/F HeadUpOK
1311  LD      M1114  ; Sheet   Feeder  AutoStep4
      MPS
      AND     T205  ; S/F     Head    Up Tm
      LD      T208  ; S/F HeadWorkVac'Det'
      OR      M6  ; S/F TestSw
      ANB
      AND<>   D24 D190  ; Sheet   Feeder  Current Position / S/F HeadSelect  Buffer
      MPS
      AND<    D24 D190  ; Sheet   Feeder  Current Position / S/F HeadSelect  Buffer
      OUT     M1137  ; Sheet   Feeder  Fwd At
      MPP
      AND>    D24 D190  ; Sheet   Feeder  Current Position / S/F HeadSelect  Buffer
      OUT     M1138  ; Sheet   Feeder  Rev At
      MRD
      LD=     D190 K14  ; S/F HeadSelect  Buffer
      AND<=   K12 D24  ; Sheet   Feeder  Current Position
      AND     M1137  ; Sheet   Feeder  Fwd At
      LD=     D190 K14  ; S/F HeadSelect  Buffer
      AND>=   K16 D24  ; Sheet   Feeder  Current Position
      AND     M1138  ; Sheet   Feeder  Rev At
      ORB
      ANB
      OUT     M1139  ; Sheet   Feeder  Slow
      MPP
      AND     M1036  ; Sheet   Feeder  CentPos'
      AND=    D24 K14  ; Sheet   Feeder  Current Position
      OUT     M1141  ; S/F ConvPositionMoveOK
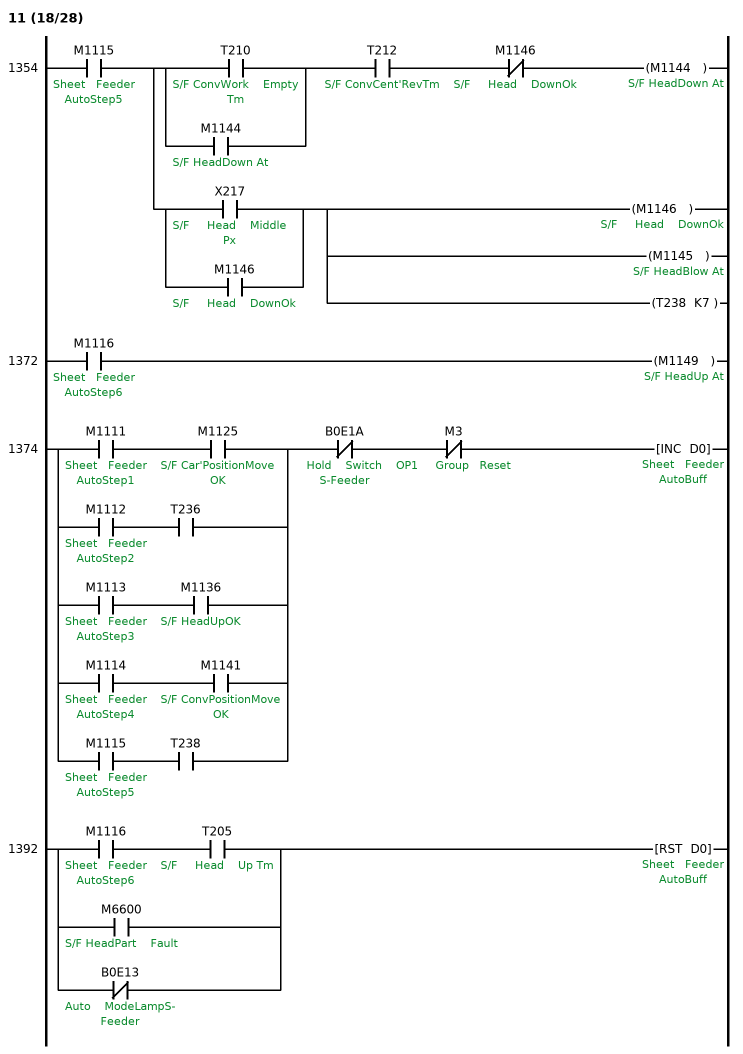
1354  LD      M1115  ; Sheet   Feeder  AutoStep5
      MPS
      LD      T210  ; S/F ConvWork    Empty Tm
      OR      M1144  ; S/F HeadDown At
      ANB
      AND     T212  ; S/F ConvCent'RevTm
      ANI     M1146  ; S/F     Head    DownOk
      OUT     M1144  ; S/F HeadDown At
      MPP
      LD      X217  ; S/F     Head    Middle  Px
      OR      M1146  ; S/F     Head    DownOk
      ANB
      OUT     M1146  ; S/F     Head    DownOk
      OUT     M1145  ; S/F HeadBlow At
      OUT     T238 K7
1372  LD      M1116  ; Sheet   Feeder  AutoStep6
      OUT     M1149  ; S/F HeadUp At
1374  LD      M1111  ; Sheet   Feeder  AutoStep1
      AND     M1125  ; S/F Car'PositionMoveOK
      LD      M1112  ; Sheet   Feeder  AutoStep2
      AND     T236
      ORB
      LD      M1113  ; Sheet   Feeder  AutoStep3
      AND     M1136  ; S/F HeadUpOK
      ORB
      LD      M1114  ; Sheet   Feeder  AutoStep4
      AND     M1141  ; S/F ConvPositionMoveOK
      ORB
      LD      M1115  ; Sheet   Feeder  AutoStep5
      AND     T238
      ORB
      ANI     B0E1A  ; Hold    Switch  S-Feeder
      ANI     M3  ; OP1     Group   Reset
      INC     D0
1392  LD      M1116  ; Sheet   Feeder  AutoStep6
      AND     T205  ; S/F     Head    Up Tm
      OR      M6600  ; S/F HeadPart    Fault
      ORI     B0E13  ; Auto    ModeLampS-Feeder
      RST     D0  ; Sheet   Feeder  AutoBuff
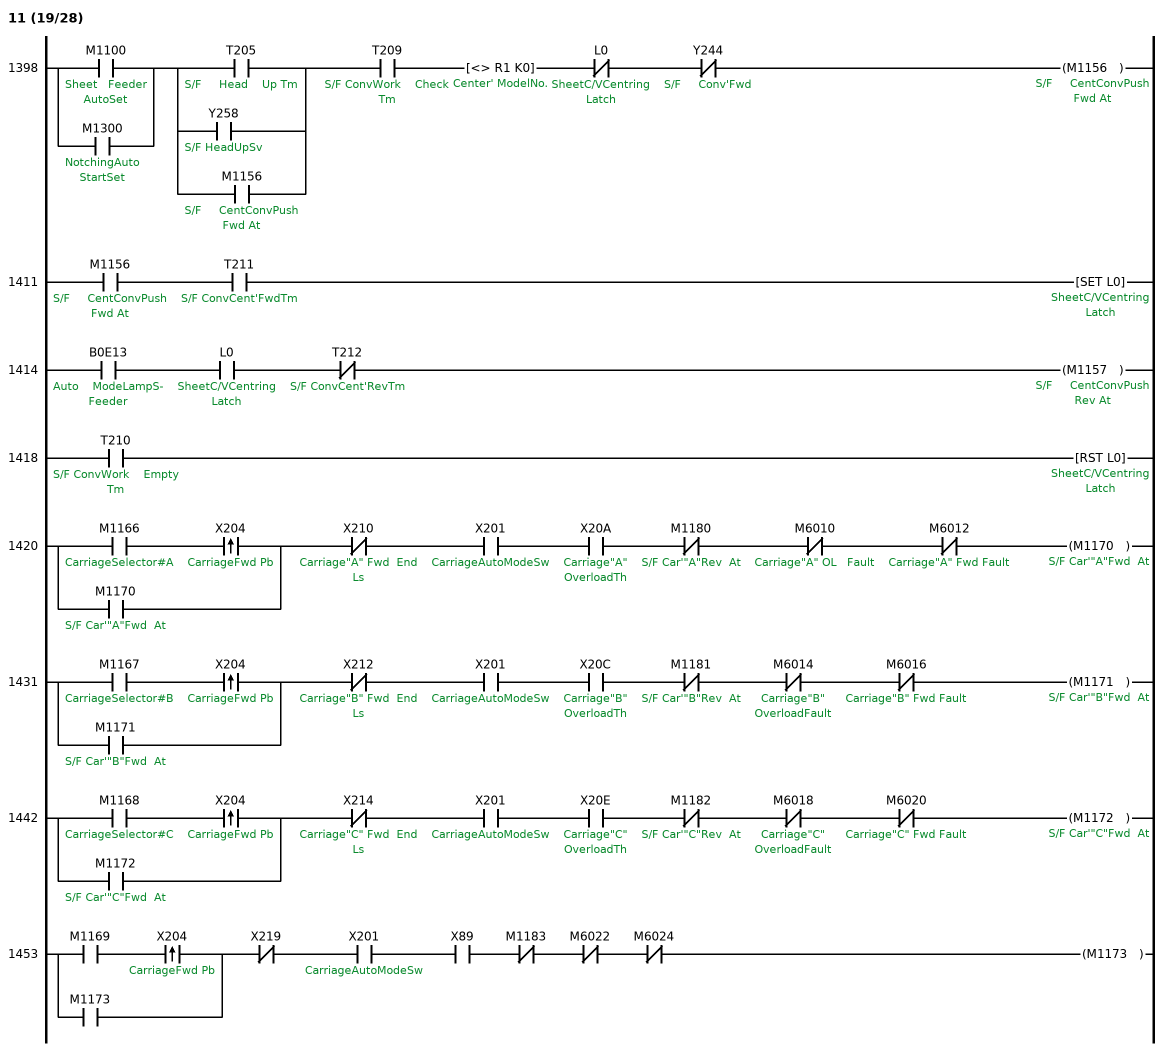
1398  LD      M1100  ; Sheet   Feeder  AutoSet
      OR      M1300  ; NotchingAuto    StartSet
      LD      T205  ; S/F     Head    Up Tm
      OR      Y258  ; S/F HeadUpSv
      OR      M1156  ; S/F     CentConvPushFwd At
      ANB
      AND     T209  ; S/F ConvWork    Check Tm
      AND<>   R1 K0  ; Center' ModelNo.
      ANI     L0  ; SheetC/VCentringLatch
      ANI     Y244  ; S/F     Conv'Fwd
      OUT     M1156  ; S/F     CentConvPushFwd At
1411  LD      M1156  ; S/F     CentConvPushFwd At
      AND     T211  ; S/F ConvCent'FwdTm
      SET     L0  ; SheetC/VCentringLatch
1414  LD      B0E13  ; Auto    ModeLampS-Feeder
      AND     L0  ; SheetC/VCentringLatch
      ANI     T212  ; S/F ConvCent'RevTm
      OUT     M1157  ; S/F     CentConvPushRev At
1418  LD      T210  ; S/F ConvWork    Empty Tm
      RST     L0  ; SheetC/VCentringLatch
1420  LD      M1166  ; CarriageSelector#A
      ANDP    X204  ; CarriageFwd Pb
      OR      M1170  ; S/F Car'"A"Fwd  At
      ANI     X210  ; Carriage"A" Fwd  End Ls
      AND     X201  ; CarriageAutoModeSw
      AND     X20A  ; Carriage"A"     OverloadTh
      ANI     M1180  ; S/F Car'"A"Rev  At
      ANI     M6010  ; Carriage"A" OL   Fault
      ANI     M6012  ; Carriage"A" Fwd Fault
      OUT     M1170  ; S/F Car'"A"Fwd  At
1431  LD      M1167  ; CarriageSelector#B
      ANDP    X204  ; CarriageFwd Pb
      OR      M1171  ; S/F Car'"B"Fwd  At
      ANI     X212  ; Carriage"B" Fwd  End Ls
      AND     X201  ; CarriageAutoModeSw
      AND     X20C  ; Carriage"B"     OverloadTh
      ANI     M1181  ; S/F Car'"B"Rev  At
      ANI     M6014  ; Carriage"B"     OverloadFault
      ANI     M6016  ; Carriage"B" Fwd Fault
      OUT     M1171  ; S/F Car'"B"Fwd  At
1442  LD      M1168  ; CarriageSelector#C
      ANDP    X204  ; CarriageFwd Pb
      OR      M1172  ; S/F Car'"C"Fwd  At
      ANI     X214  ; Carriage"C" Fwd  End Ls
      AND     X201  ; CarriageAutoModeSw
      AND     X20E  ; Carriage"C"     OverloadTh
      ANI     M1182  ; S/F Car'"C"Rev  At
      ANI     M6018  ; Carriage"C"     OverloadFault
      ANI     M6020  ; Carriage"C" Fwd Fault
      OUT     M1172  ; S/F Car'"C"Fwd  At
1453  LD      M1169
      ANDP    X204  ; CarriageFwd Pb
      OR      M1173
      ANI     X219
      AND     X201  ; CarriageAutoModeSw
      AND     X89
      ANI     M1183
      ANI     M6022
      ANI     M6024
      OUT     M1173
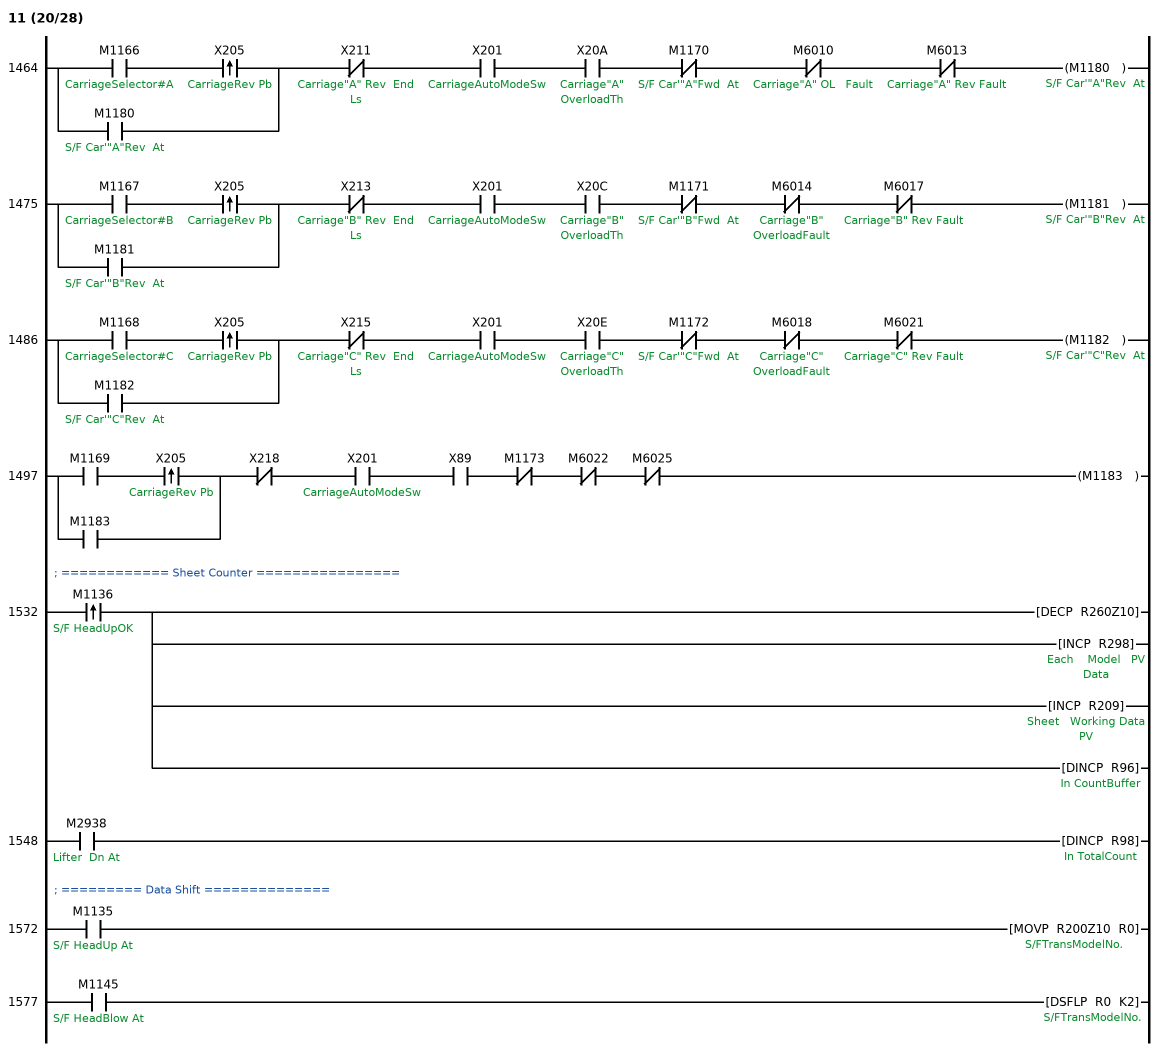
1464  LD      M1166  ; CarriageSelector#A
      ANDP    X205  ; CarriageRev Pb
      OR      M1180  ; S/F Car'"A"Rev  At
      ANI     X211  ; Carriage"A" Rev  End Ls
      AND     X201  ; CarriageAutoModeSw
      AND     X20A  ; Carriage"A"     OverloadTh
      ANI     M1170  ; S/F Car'"A"Fwd  At
      ANI     M6010  ; Carriage"A" OL   Fault
      ANI     M6013  ; Carriage"A" Rev Fault
      OUT     M1180  ; S/F Car'"A"Rev  At
1475  LD      M1167  ; CarriageSelector#B
      ANDP    X205  ; CarriageRev Pb
      OR      M1181  ; S/F Car'"B"Rev  At
      ANI     X213  ; Carriage"B" Rev  End Ls
      AND     X201  ; CarriageAutoModeSw
      AND     X20C  ; Carriage"B"     OverloadTh
      ANI     M1171  ; S/F Car'"B"Fwd  At
      ANI     M6014  ; Carriage"B"     OverloadFault
      ANI     M6017  ; Carriage"B" Rev Fault
      OUT     M1181  ; S/F Car'"B"Rev  At
1486  LD      M1168  ; CarriageSelector#C
      ANDP    X205  ; CarriageRev Pb
      OR      M1182  ; S/F Car'"C"Rev  At
      ANI     X215  ; Carriage"C" Rev  End Ls
      AND     X201  ; CarriageAutoModeSw
      AND     X20E  ; Carriage"C"     OverloadTh
      ANI     M1172  ; S/F Car'"C"Fwd  At
      ANI     M6018  ; Carriage"C"     OverloadFault
      ANI     M6021  ; Carriage"C" Rev Fault
      OUT     M1182  ; S/F Car'"C"Rev  At
1497  LD      M1169
      ANDP    X205  ; CarriageRev Pb
      OR      M1183
      ANI     X218
      AND     X201  ; CarriageAutoModeSw
      AND     X89
      ANI     M1173
      ANI     M6022
      ANI     M6025
      OUT     M1183
; ============ Sheet Counter ================
1532  LDP     M1136  ; S/F HeadUpOK
      DECP    R260Z10
      INCP    R298
      INCP    R209
      DINCP   R96  ; In CountBuffer
1548  LD      M2938  ; Lifter  Dn At
      DINCP   R98  ; In TotalCount
; ========= Data Shift ==============
1572  LD      M1135  ; S/F HeadUp At
      MOVP    R200Z10 R0  ; S/FTransModelNo.
1577  LD      M1145  ; S/F HeadBlow At
      DSFLP   R0 K2
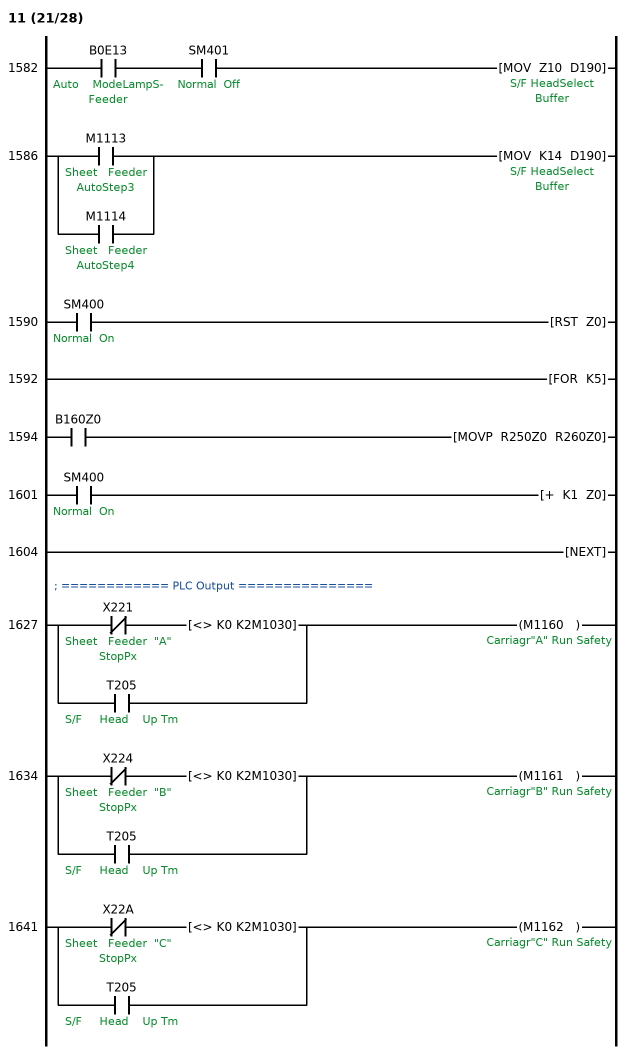
1582  LD      B0E13  ; Auto    ModeLampS-Feeder
      AND     SM401  ; Normal  Off
      MOV     Z10 D190
1586  LD      M1113  ; Sheet   Feeder  AutoStep3
      OR      M1114  ; Sheet   Feeder  AutoStep4
      MOV     K14 D190
1590  LD      SM400  ; Normal  On
      RST     Z0
1592  FOR     K5
1594  LD      B160Z0
      MOVP    R250Z0 R260Z0
1601  LD      SM400  ; Normal  On
      +       K1 Z0
1604  NEXT
; ============ PLC Output ===============
1627  LDI     X221  ; Sheet   Feeder  "A" StopPx
      AND<>   K0 K2M1030  ; Sheet   Feeder  "A" Pos'
      OR      T205  ; S/F     Head    Up Tm
      OUT     M1160  ; Carriagr"A" Run Safety
1634  LDI     X224  ; Sheet   Feeder  "B" StopPx
      AND<>   K0 K2M1030  ; Sheet   Feeder  "A" Pos'
      OR      T205  ; S/F     Head    Up Tm
      OUT     M1161  ; Carriagr"B" Run Safety
1641  LDI     X22A  ; Sheet   Feeder  "C" StopPx
      AND<>   K0 K2M1030  ; Sheet   Feeder  "A" Pos'
      OR      T205  ; S/F     Head    Up Tm
      OUT     M1162  ; Carriagr"C" Run Safety
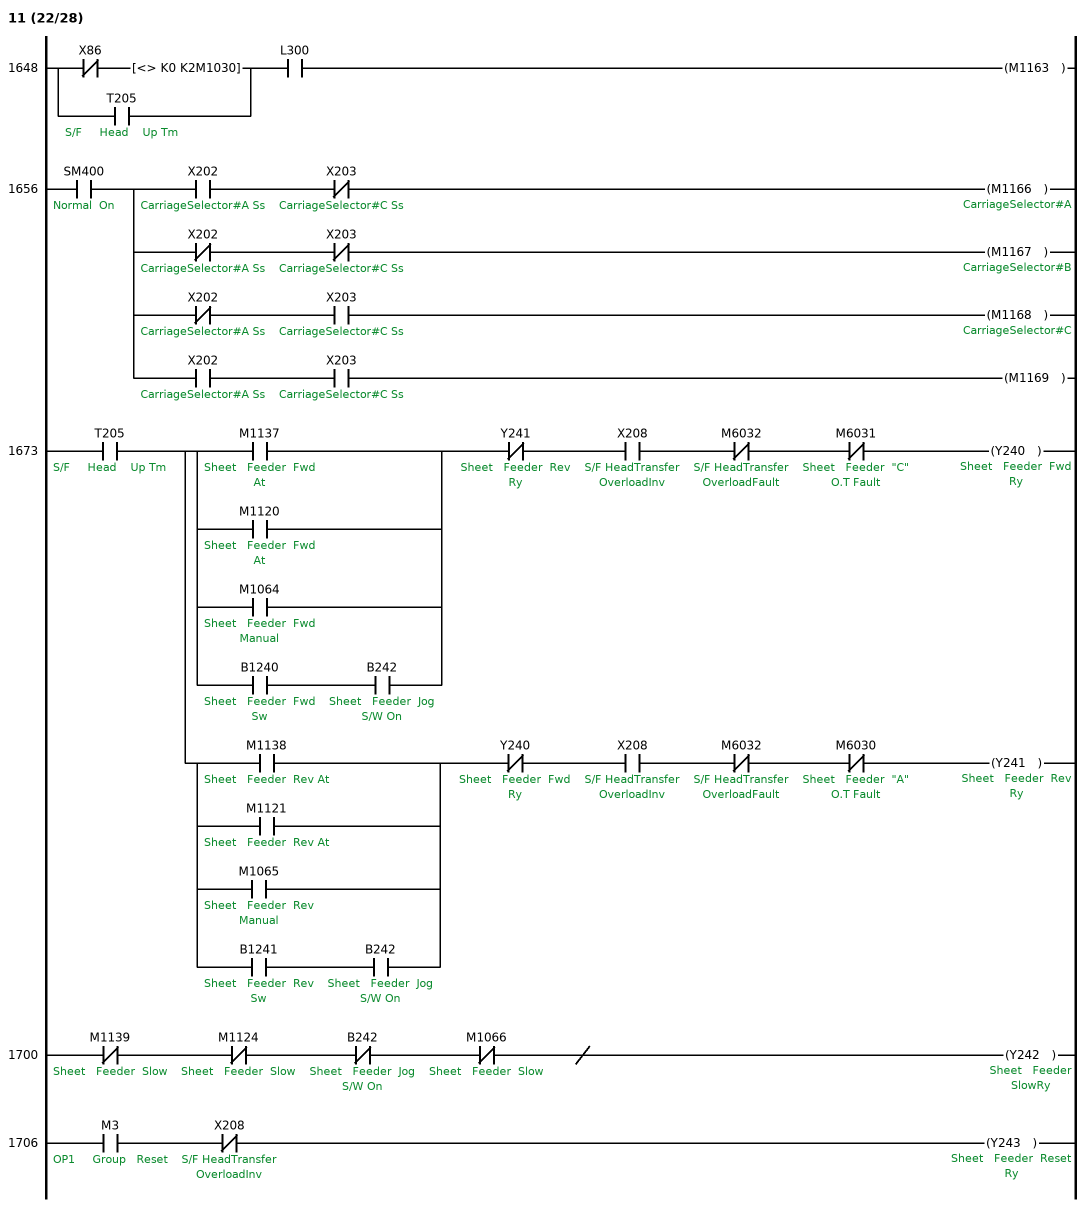
1648  LDI     X86
      AND<>   K0 K2M1030  ; Sheet   Feeder  "A" Pos'
      OR      T205  ; S/F     Head    Up Tm
      AND     L300
      OUT     M1163
1656  LD      SM400  ; Normal  On
      MPS
      AND     X202  ; CarriageSelector#A Ss
      ANI     X203  ; CarriageSelector#C Ss
      OUT     M1166  ; CarriageSelector#A
      MRD
      ANI     X202  ; CarriageSelector#A Ss
      ANI     X203  ; CarriageSelector#C Ss
      OUT     M1167  ; CarriageSelector#B
      MRD
      ANI     X202  ; CarriageSelector#A Ss
      AND     X203  ; CarriageSelector#C Ss
      OUT     M1168  ; CarriageSelector#C
      MPP
      AND     X202  ; CarriageSelector#A Ss
      AND     X203  ; CarriageSelector#C Ss
      OUT     M1169
1673  LD      T205  ; S/F     Head    Up Tm
      MPS
      LD      M1137  ; Sheet   Feeder  Fwd At
      OR      M1120  ; Sheet   Feeder  Fwd At
      OR      M1064  ; Sheet   Feeder  Fwd     Manual
      LD      B1240  ; Sheet   Feeder  Fwd Sw
      AND     B242  ; Sheet   Feeder  Jog S/W On
      ORB
      ANB
      ANI     Y241  ; Sheet   Feeder  Rev Ry
      AND     X208  ; S/F HeadTransferOverloadInv
      ANI     M6032  ; S/F HeadTransferOverloadFault
      ANI     M6031  ; Sheet   Feeder  "C" O.T Fault
      OUT     Y240  ; Sheet   Feeder  Fwd Ry
      MPP
      LD      M1138  ; Sheet   Feeder  Rev At
      OR      M1121  ; Sheet   Feeder  Rev At
      OR      M1065  ; Sheet   Feeder  Rev     Manual
      LD      B1241  ; Sheet   Feeder  Rev Sw
      AND     B242  ; Sheet   Feeder  Jog S/W On
      ORB
      ANB
      ANI     Y240  ; Sheet   Feeder  Fwd Ry
      AND     X208  ; S/F HeadTransferOverloadInv
      ANI     M6032  ; S/F HeadTransferOverloadFault
      ANI     M6030  ; Sheet   Feeder  "A" O.T Fault
      OUT     Y241  ; Sheet   Feeder  Rev Ry
1700  LDI     M1139  ; Sheet   Feeder  Slow
      ANI     M1124  ; Sheet   Feeder  Slow
      ANI     B242  ; Sheet   Feeder  Jog S/W On
      ANI     M1066  ; Sheet   Feeder  Slow
      INV
      OUT     Y242  ; Sheet   Feeder  SlowRy
1706  LD      M3  ; OP1     Group   Reset
      ANI     X208  ; S/F HeadTransferOverloadInv
      OUT     Y243  ; Sheet   Feeder  Reset Ry
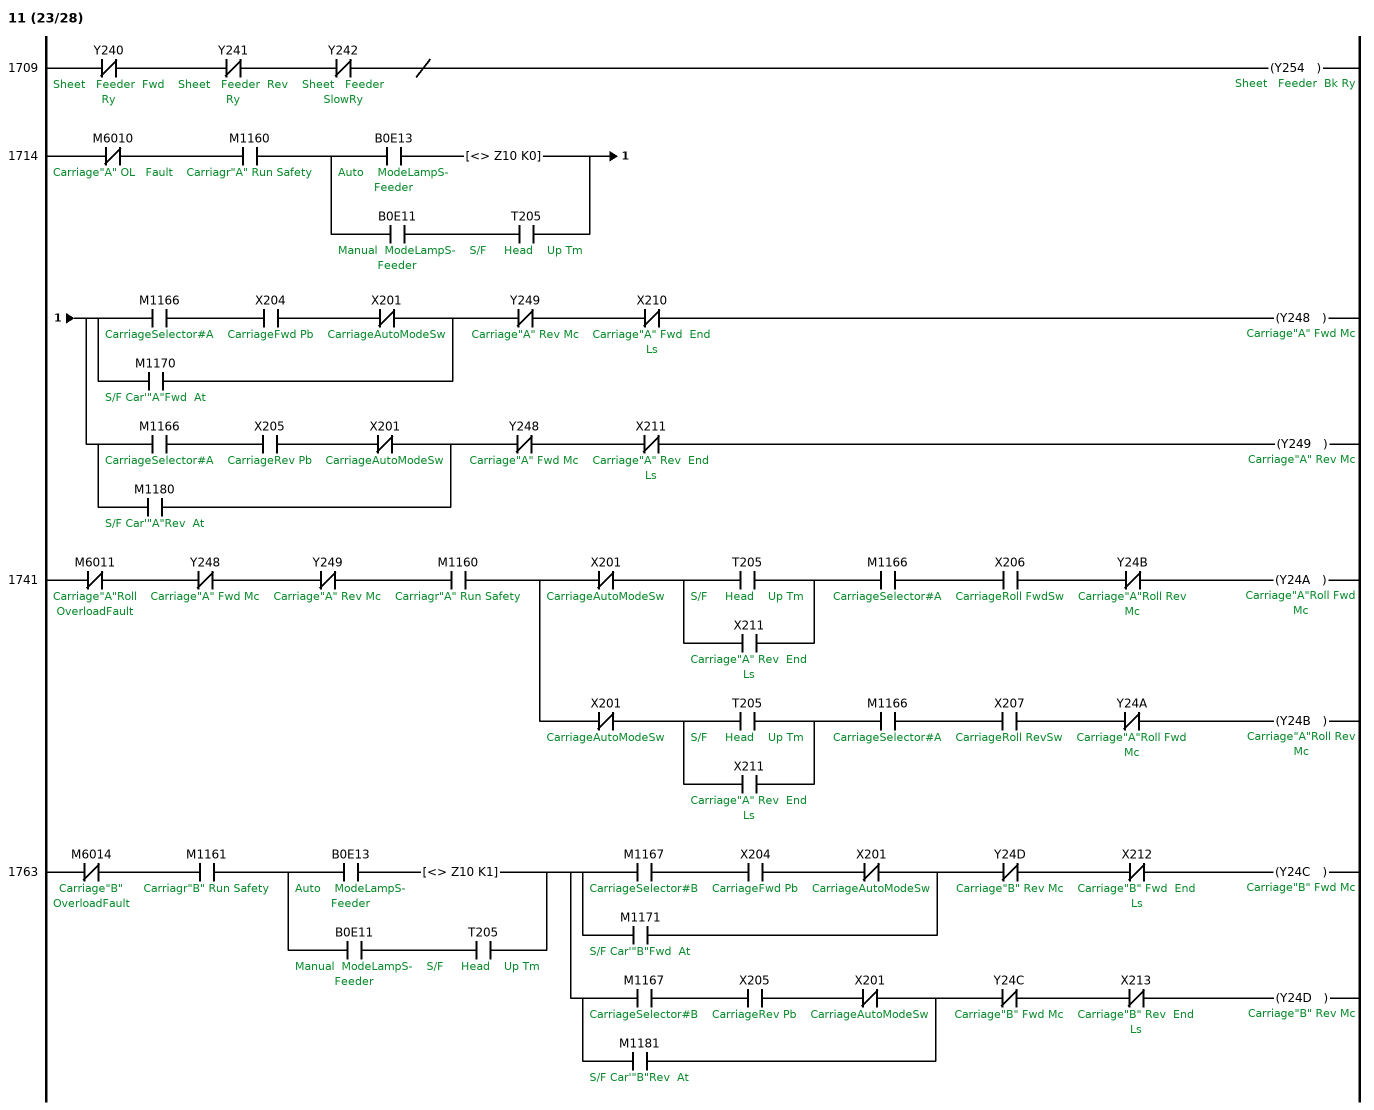
1709  LDI     Y240  ; Sheet   Feeder  Fwd Ry
      ANI     Y241  ; Sheet   Feeder  Rev Ry
      ANI     Y242  ; Sheet   Feeder  SlowRy
      INV
      OUT     Y254  ; Sheet   Feeder  Bk Ry
1714  LDI     M6010  ; Carriage"A" OL   Fault
      AND     M1160  ; Carriagr"A" Run Safety
      LD      B0E13  ; Auto    ModeLampS-Feeder
      AND<>   Z10 K0
      LD      B0E11  ; Manual  ModeLampS-Feeder
      AND     T205  ; S/F     Head    Up Tm
      ORB
      ANB
      MPS
      LD      M1166  ; CarriageSelector#A
      AND     X204  ; CarriageFwd Pb
      ANI     X201  ; CarriageAutoModeSw
      OR      M1170  ; S/F Car'"A"Fwd  At
      ANB
      ANI     Y249  ; Carriage"A" Rev Mc
      ANI     X210  ; Carriage"A" Fwd  End Ls
      OUT     Y248  ; Carriage"A" Fwd Mc
      MPP
      LD      M1166  ; CarriageSelector#A
      AND     X205  ; CarriageRev Pb
      ANI     X201  ; CarriageAutoModeSw
      OR      M1180  ; S/F Car'"A"Rev  At
      ANB
      ANI     Y248  ; Carriage"A" Fwd Mc
      ANI     X211  ; Carriage"A" Rev  End Ls
      OUT     Y249  ; Carriage"A" Rev Mc
1741  LDI     M6011  ; Carriage"A"Roll OverloadFault
      ANI     Y248  ; Carriage"A" Fwd Mc
      ANI     Y249  ; Carriage"A" Rev Mc
      AND     M1160  ; Carriagr"A" Run Safety
      MPS
      ANI     X201  ; CarriageAutoModeSw
      LD      T205  ; S/F     Head    Up Tm
      OR      X211  ; Carriage"A" Rev  End Ls
      ANB
      AND     M1166  ; CarriageSelector#A
      AND     X206  ; CarriageRoll FwdSw
      ANI     Y24B  ; Carriage"A"Roll Rev Mc
      OUT     Y24A  ; Carriage"A"Roll Fwd Mc
      MPP
      ANI     X201  ; CarriageAutoModeSw
      LD      T205  ; S/F     Head    Up Tm
      OR      X211  ; Carriage"A" Rev  End Ls
      ANB
      AND     M1166  ; CarriageSelector#A
      AND     X207  ; CarriageRoll RevSw
      ANI     Y24A  ; Carriage"A"Roll Fwd Mc
      OUT     Y24B  ; Carriage"A"Roll Rev Mc
1763  LDI     M6014  ; Carriage"B"     OverloadFault
      AND     M1161  ; Carriagr"B" Run Safety
      LD      B0E13  ; Auto    ModeLampS-Feeder
      AND<>   Z10 K1
      LD      B0E11  ; Manual  ModeLampS-Feeder
      AND     T205  ; S/F     Head    Up Tm
      ORB
      ANB
      MPS
      LD      M1167  ; CarriageSelector#B
      AND     X204  ; CarriageFwd Pb
      ANI     X201  ; CarriageAutoModeSw
      OR      M1171  ; S/F Car'"B"Fwd  At
      ANB
      ANI     Y24D  ; Carriage"B" Rev Mc
      ANI     X212  ; Carriage"B" Fwd  End Ls
      OUT     Y24C  ; Carriage"B" Fwd Mc
      MPP
      LD      M1167  ; CarriageSelector#B
      AND     X205  ; CarriageRev Pb
      ANI     X201  ; CarriageAutoModeSw
      OR      M1181  ; S/F Car'"B"Rev  At
      ANB
      ANI     Y24C  ; Carriage"B" Fwd Mc
      ANI     X213  ; Carriage"B" Rev  End Ls
      OUT     Y24D  ; Carriage"B" Rev Mc
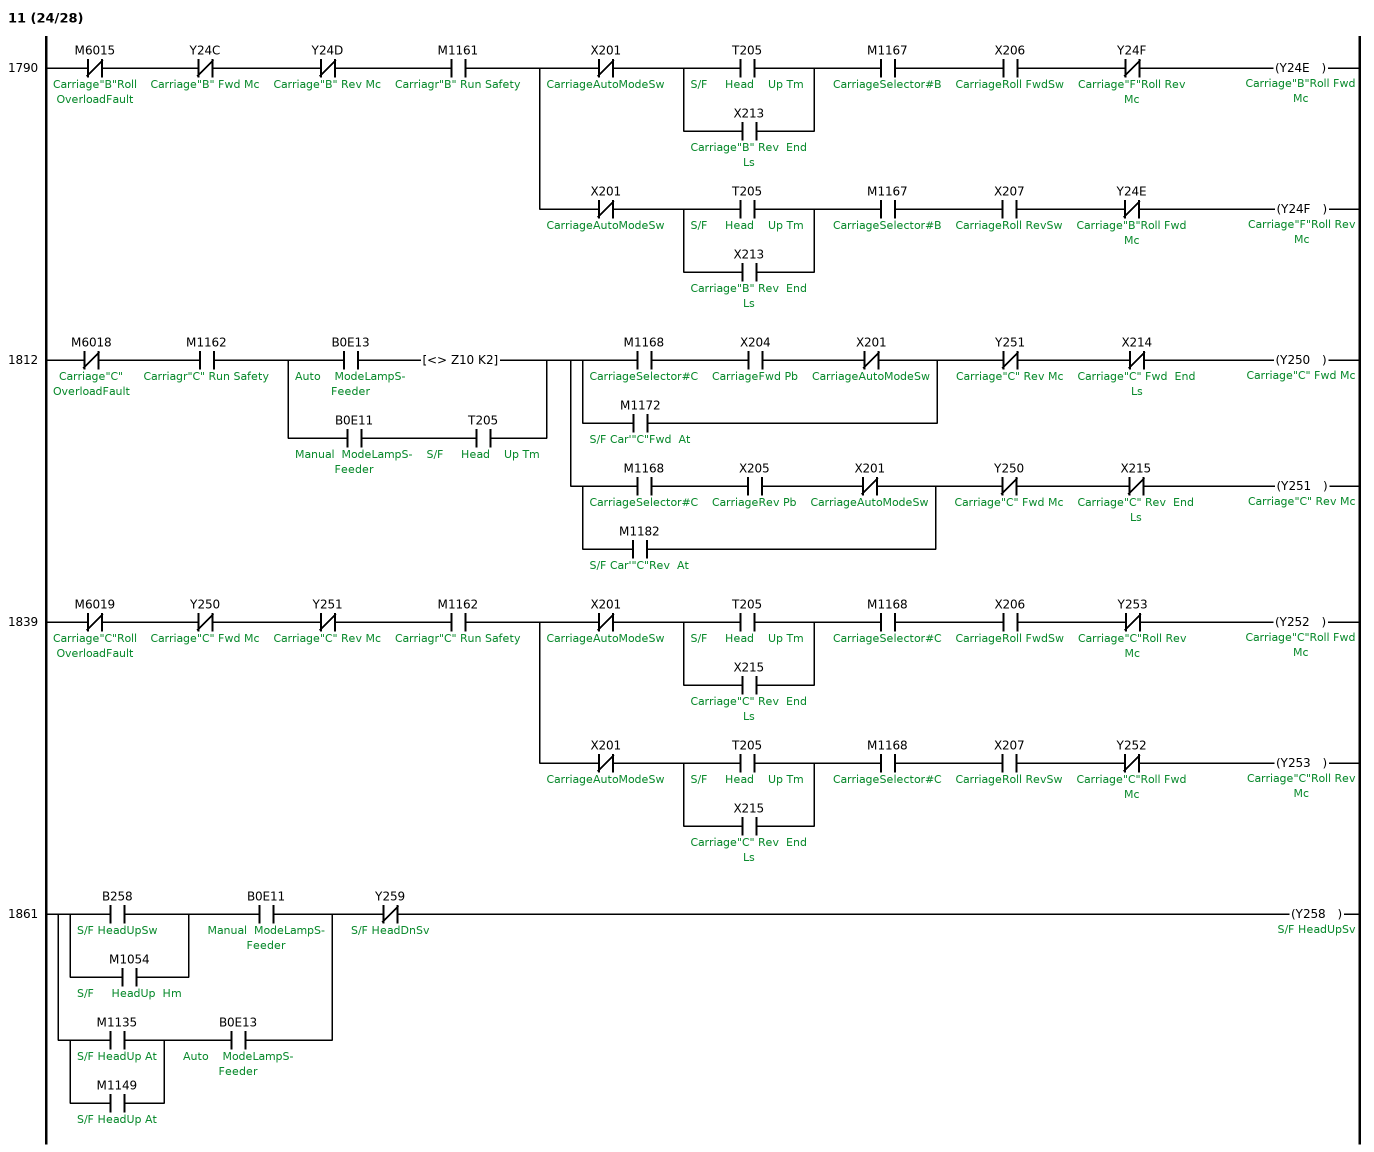
1790  LDI     M6015  ; Carriage"B"Roll OverloadFault
      ANI     Y24C  ; Carriage"B" Fwd Mc
      ANI     Y24D  ; Carriage"B" Rev Mc
      AND     M1161  ; Carriagr"B" Run Safety
      MPS
      ANI     X201  ; CarriageAutoModeSw
      LD      T205  ; S/F     Head    Up Tm
      OR      X213  ; Carriage"B" Rev  End Ls
      ANB
      AND     M1167  ; CarriageSelector#B
      AND     X206  ; CarriageRoll FwdSw
      ANI     Y24F  ; Carriage"F"Roll Rev Mc
      OUT     Y24E  ; Carriage"B"Roll Fwd Mc
      MPP
      ANI     X201  ; CarriageAutoModeSw
      LD      T205  ; S/F     Head    Up Tm
      OR      X213  ; Carriage"B" Rev  End Ls
      ANB
      AND     M1167  ; CarriageSelector#B
      AND     X207  ; CarriageRoll RevSw
      ANI     Y24E  ; Carriage"B"Roll Fwd Mc
      OUT     Y24F  ; Carriage"F"Roll Rev Mc
1812  LDI     M6018  ; Carriage"C"     OverloadFault
      AND     M1162  ; Carriagr"C" Run Safety
      LD      B0E13  ; Auto    ModeLampS-Feeder
      AND<>   Z10 K2
      LD      B0E11  ; Manual  ModeLampS-Feeder
      AND     T205  ; S/F     Head    Up Tm
      ORB
      ANB
      MPS
      LD      M1168  ; CarriageSelector#C
      AND     X204  ; CarriageFwd Pb
      ANI     X201  ; CarriageAutoModeSw
      OR      M1172  ; S/F Car'"C"Fwd  At
      ANB
      ANI     Y251  ; Carriage"C" Rev Mc
      ANI     X214  ; Carriage"C" Fwd  End Ls
      OUT     Y250  ; Carriage"C" Fwd Mc
      MPP
      LD      M1168  ; CarriageSelector#C
      AND     X205  ; CarriageRev Pb
      ANI     X201  ; CarriageAutoModeSw
      OR      M1182  ; S/F Car'"C"Rev  At
      ANB
      ANI     Y250  ; Carriage"C" Fwd Mc
      ANI     X215  ; Carriage"C" Rev  End Ls
      OUT     Y251  ; Carriage"C" Rev Mc
1839  LDI     M6019  ; Carriage"C"Roll OverloadFault
      ANI     Y250  ; Carriage"C" Fwd Mc
      ANI     Y251  ; Carriage"C" Rev Mc
      AND     M1162  ; Carriagr"C" Run Safety
      MPS
      ANI     X201  ; CarriageAutoModeSw
      LD      T205  ; S/F     Head    Up Tm
      OR      X215  ; Carriage"C" Rev  End Ls
      ANB
      AND     M1168  ; CarriageSelector#C
      AND     X206  ; CarriageRoll FwdSw
      ANI     Y253  ; Carriage"C"Roll Rev Mc
      OUT     Y252  ; Carriage"C"Roll Fwd Mc
      MPP
      ANI     X201  ; CarriageAutoModeSw
      LD      T205  ; S/F     Head    Up Tm
      OR      X215  ; Carriage"C" Rev  End Ls
      ANB
      AND     M1168  ; CarriageSelector#C
      AND     X207  ; CarriageRoll RevSw
      ANI     Y252  ; Carriage"C"Roll Fwd Mc
      OUT     Y253  ; Carriage"C"Roll Rev Mc
1861  LD      B258  ; S/F HeadUpSw
      OR      M1054  ; S/F     HeadUp  Hm
      AND     B0E11  ; Manual  ModeLampS-Feeder
      LD      M1135  ; S/F HeadUp At
      OR      M1149  ; S/F HeadUp At
      AND     B0E13  ; Auto    ModeLampS-Feeder
      ORB
      ANI     Y259  ; S/F HeadDnSv
      OUT     Y258  ; S/F HeadUpSv
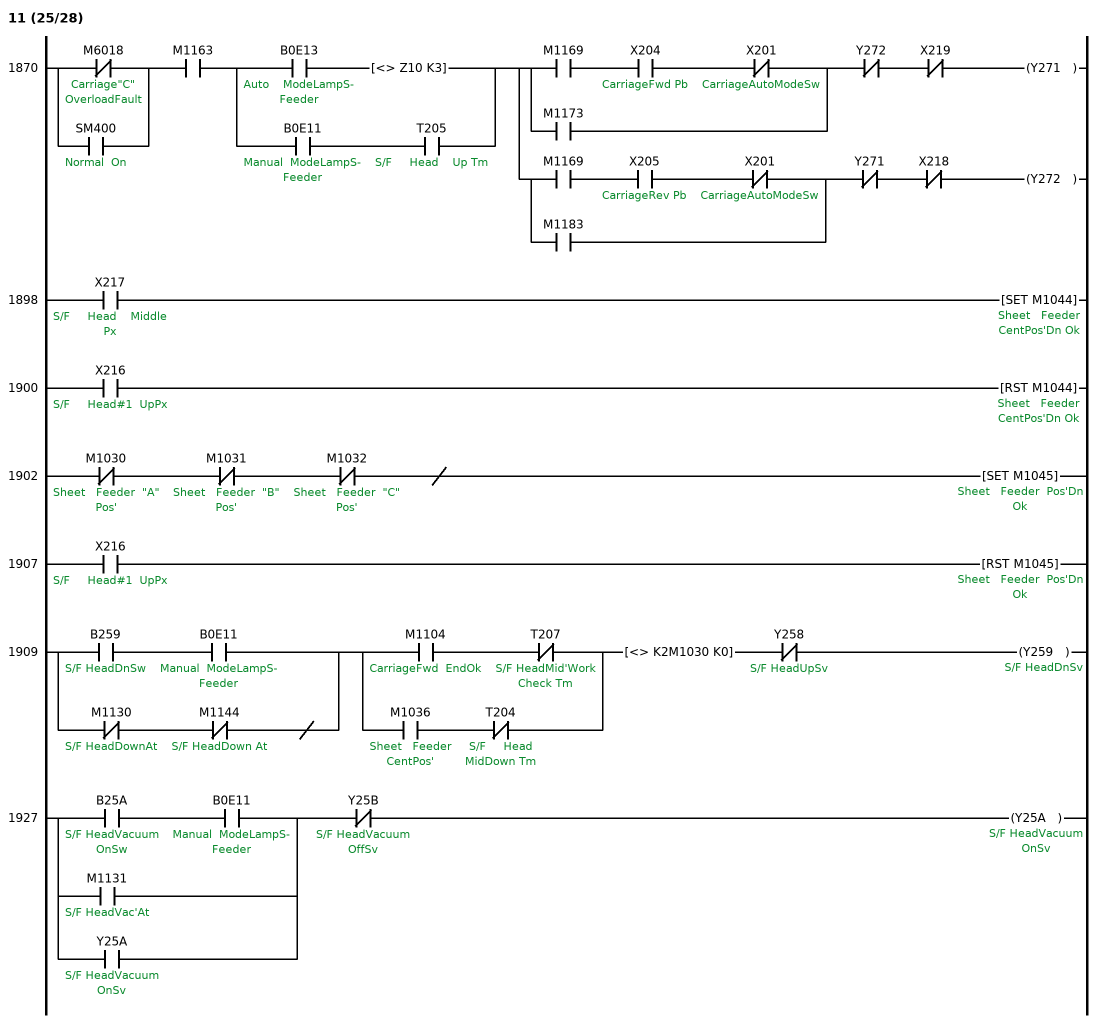
1870  LDI     M6018  ; Carriage"C"     OverloadFault
      OR      SM400  ; Normal  On
      AND     M1163
      LD      B0E13  ; Auto    ModeLampS-Feeder
      AND<>   Z10 K3
      LD      B0E11  ; Manual  ModeLampS-Feeder
      AND     T205  ; S/F     Head    Up Tm
      ORB
      ANB
      MPS
      LD      M1169
      AND     X204  ; CarriageFwd Pb
      ANI     X201  ; CarriageAutoModeSw
      OR      M1173
      ANB
      ANI     Y272
      ANI     X219
      OUT     Y271
      MPP
      LD      M1169
      AND     X205  ; CarriageRev Pb
      ANI     X201  ; CarriageAutoModeSw
      OR      M1183
      ANB
      ANI     Y271
      ANI     X218
      OUT     Y272
1898  LD      X217  ; S/F     Head    Middle  Px
      SET     M1044  ; Sheet   Feeder  CentPos'Dn Ok
1900  LD      X216  ; S/F     Head#1  UpPx
      RST     M1044  ; Sheet   Feeder  CentPos'Dn Ok
1902  LDI     M1030  ; Sheet   Feeder  "A" Pos'
      ANI     M1031  ; Sheet   Feeder  "B" Pos'
      ANI     M1032  ; Sheet   Feeder  "C" Pos'
      INV
      SET     M1045  ; Sheet   Feeder  Pos'Dn  Ok
1907  LD      X216  ; S/F     Head#1  UpPx
      RST     M1045  ; Sheet   Feeder  Pos'Dn  Ok
1909  LD      B259  ; S/F HeadDnSw
      AND     B0E11  ; Manual  ModeLampS-Feeder
      LDI     M1130  ; S/F HeadDownAt
      ANI     M1144  ; S/F HeadDown At
      INV
      ORB
      LD      M1104  ; CarriageFwd  EndOk
      ANI     T207  ; S/F HeadMid'WorkCheck Tm
      LD      M1036  ; Sheet   Feeder  CentPos'
      ANI     T204  ; S/F     Head    MidDown Tm
      ORB
      ANB
      AND<>   K2M1030 K0  ; Sheet   Feeder  "A" Pos'
      ANI     Y258  ; S/F HeadUpSv
      OUT     Y259  ; S/F HeadDnSv
1927  LD      B25A  ; S/F HeadVacuum  OnSw
      AND     B0E11  ; Manual  ModeLampS-Feeder
      OR      M1131  ; S/F HeadVac'At
      OR      Y25A  ; S/F HeadVacuum  OnSv
      ANI     Y25B  ; S/F HeadVacuum  OffSv
      OUT     Y25A  ; S/F HeadVacuum  OnSv
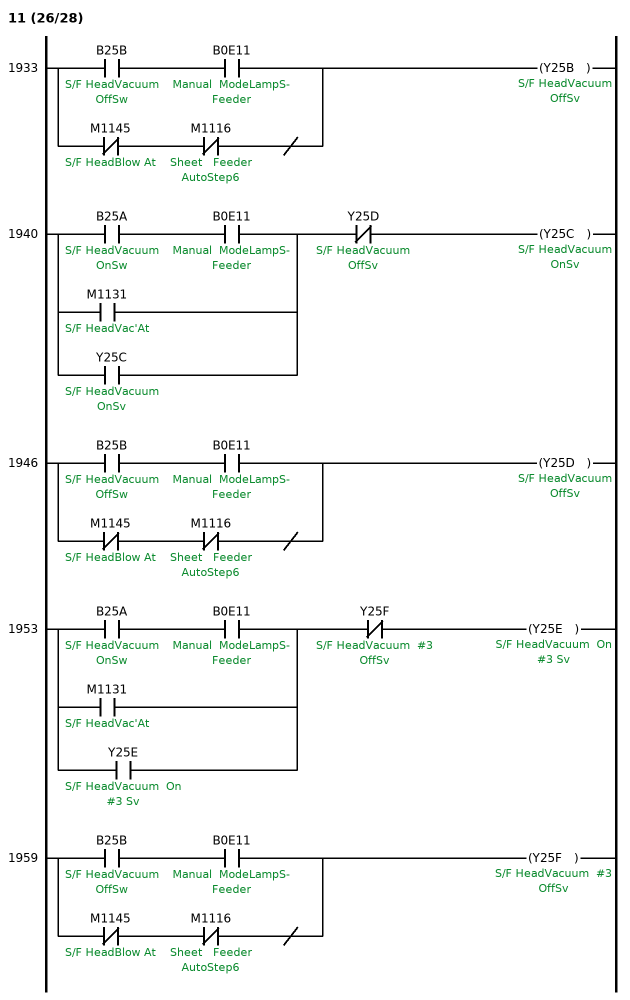
1933  LD      B25B  ; S/F HeadVacuum  OffSw
      AND     B0E11  ; Manual  ModeLampS-Feeder
      LDI     M1145  ; S/F HeadBlow At
      ANI     M1116  ; Sheet   Feeder  AutoStep6
      INV
      ORB
      OUT     Y25B  ; S/F HeadVacuum  OffSv
1940  LD      B25A  ; S/F HeadVacuum  OnSw
      AND     B0E11  ; Manual  ModeLampS-Feeder
      OR      M1131  ; S/F HeadVac'At
      OR      Y25C  ; S/F HeadVacuum  OnSv
      ANI     Y25D  ; S/F HeadVacuum  OffSv
      OUT     Y25C  ; S/F HeadVacuum  OnSv
1946  LD      B25B  ; S/F HeadVacuum  OffSw
      AND     B0E11  ; Manual  ModeLampS-Feeder
      LDI     M1145  ; S/F HeadBlow At
      ANI     M1116  ; Sheet   Feeder  AutoStep6
      INV
      ORB
      OUT     Y25D  ; S/F HeadVacuum  OffSv
1953  LD      B25A  ; S/F HeadVacuum  OnSw
      AND     B0E11  ; Manual  ModeLampS-Feeder
      OR      M1131  ; S/F HeadVac'At
      OR      Y25E  ; S/F HeadVacuum  On #3 Sv
      ANI     Y25F  ; S/F HeadVacuum  #3 OffSv
      OUT     Y25E  ; S/F HeadVacuum  On #3 Sv
1959  LD      B25B  ; S/F HeadVacuum  OffSw
      AND     B0E11  ; Manual  ModeLampS-Feeder
      LDI     M1145  ; S/F HeadBlow At
      ANI     M1116  ; Sheet   Feeder  AutoStep6
      INV
      ORB
      OUT     Y25F  ; S/F HeadVacuum  #3 OffSv
